# B&R Automation Studio project VInRoS_BaR_AS_Program
Automation Studio 4.12.5.95 SP; technology packages: mapp 5.24.2, mappCockpit 5.24.2, mappMotion 5.26.1, mappView 5.24.2

## Configuration Config_5APC2100

CPU 5APC2100.BY48-000, AutomationRuntime B4.83, Build 4.1.2, Safety 1.10, Vc V4.72.6

### Task classes (Cpu.sw)
```
Cyclic#1 (cycle 2000 us, tolerance 0 us):
  T_MECH_1 <- T_MECH_1.prg
  T_MECH_2 <- T_MECH_2.prg
  T_MECH_3 <- T_MECH_3.prg
Cyclic#2 (cycle 4000 us, tolerance 0 us):
  T_ROB_1 <- T_ROB_1.prg
  T_ROB_2_L <- T_ROB_2_L.prg
  T_ROB_2_R <- T_ROB_2_R.prg
Cyclic#3 (cycle 10000 us, tolerance 0 us):
  T_EX600 <- T_EX600.prg
DataObjects: assl1, McAcpSys
NcDataObjects: McDriveLog
Binaries: arsvcreg, FWRules, McAcpSim, mvLoader, mCoWebSc, McAcpDrv, TCData, udbdef, arflatprv, arcoal, iomap, asfw, Settings, Role, Cfg_mMot, sysconf, asnxdb1, arconfig, ashwac, ashwd, User, asnxdb2
Libraries: McBase, CoTrace, AsZip, FileIO, runtime, AsSafety, standard, DataObj, AsXml, astime, McAxis, McAcpAx, McAcpPar, McAxGroup, MpAxis, MpBase, arssl, powerlnk, asepl
```

### Hardware
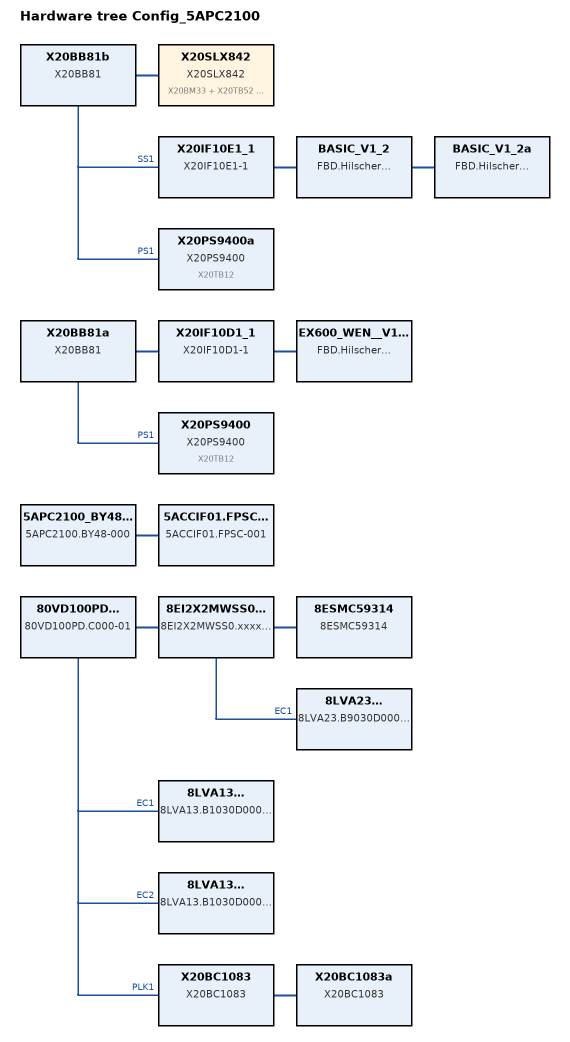
```
5ACCIF01.FPSC-001 : 5ACCIF01.FPSC-001 v1.9.1.0  [SL -> 5APC2100_BY48_000.SL1]
  Connector IF1:
    DNAConfiguration = manual
    Channel1
    ChannelID1 = McAcpBroadcast
    ChannelType1 = OCTET[128]
5APC2100_BY48_000 : 5APC2100.BY48-000 v2.1.1.0
  Connector IF3:
    AssignedOperatingSystem = ARemb
    ActivateDevice = 1
  Connector IF4:
    AssignedOperatingSystem = GPOS
  Connector IF7:
    OperatingSystem = ARemb
    ActivateDevice = 1
  Connector IF5:
    AssignedOperatingSystem = ARemb
  Connector IF6:
    AssignedOperatingSystem = GPOS
  ConfigurationID = BR_AS_I4C_Program_Config_5APC2100
  TimerDeviceType = EPLX2X
  TimerDevice = 5ACCIF01.FPSC-001.IF1
  TaskClassIdleTime = 2000
  Cyclic1Duration = 2000
  Cyclic1Tolerance = 0
  Cyclic2Duration = 4000
  Cyclic2Tolerance = 0
  Cyclic3Duration = 10000
  Cyclic3Tolerance = 0
  ActivateOpcUa = 1
  OpcUaInformationModels_PV_Version = 1
  ActivateHypervisor = 1
  ARembDramSizeInMb = 2000
80VD100PD.C000-01 : 80VD100PD.C000-01 v2.5.0.0  [PLK1 -> X20BC1083.PLK1 (NodeNumber=3) [Cable Type=PowerlinkCable, Length=10, Version=1.0.0.3]; PLK2 -> 8EI2X2MWSS0.xxxx-1.PLK1 (NodeNumber=3) [Cable Type=PowerlinkCable, Length=10, Version=1.0.0.3]; EC1 -> 8LVA13.B1030D000-0.EC; EC2 -> 8LVA13.B1030D000-0a.EC; MT2 -> 8LVA13.B1030D000-0a.MT]
  EnableDNA = on
  EPL_DNA_HubPort = 1
  DriveConfiguration/Module:
    McAcoposTypeID = AcoposMicroDConfig
    ActivateACOPOSSimulationOnPLC = 0
  DriveConfiguration/Channel[1]/RealAxis:
    AxisReference = gAxis_Mech_01
    MechanicalElementsIsInvisible = 0
  DriveConfiguration/Channel[1]/RealAxis/MechanicalElements/Gearbox:
    InputIsReadOnly = 0
    Input = 1
    OutputIsReadOnly = 0
    Output = 1
  DriveConfiguration/Channel[1]/RealAxis/MechanicalElements/RotaryToLinearTransformation:
    ReferenceDistanceIsReadOnly = 0
    ReferenceDistance = 54
  DriveConfiguration/Channel[1]/RealAxis/Controller:
    ModeIsReadOnly = 0
    Mode = PositionControllerWithTorqueFeedForward
  DriveConfiguration/Channel[1]/RealAxis/Controller/Mode/Position:
    ProportionalGainIsReadOnly = 0
    ProportionalGain = 279.0
    IntegrationTimeIsReadOnly = 0
    IntegrationTime = 0.000000
    TotalDelayTime = 0.0004
  DriveConfiguration/Channel[1]/RealAxis/Controller/Mode/Speed:
    ProportionalGainIsReadOnly = 0
    ProportionalGain = 0.25
    IntegrationTimeIsReadOnly = 0
    IntegrationTime = 0.000000
    FilterTimeIsReadOnly = 0
    FilterTime = 0.000000
  DriveConfiguration/Channel[1]/RealAxis/Controller/Mode:
    FeedForwardIsReadOnly = 0
    FeedForward = Standard
  DriveConfiguration/Channel[1]/RealAxis/Controller/Mode/FeedForward:
    TorqueLoad = 0.000000
    TorquePositive = 0.0326912
    TorqueNegative = 0.03062093
    SpeedTorqueFactor = 0.002517087
    Inertia = 0.00005712706
    AccelerationFilterTime = 0.000000
  DriveConfiguration/Channel[1]/RealAxis/Controller/Mode/LoopFilters:
    LoopFilterXIsReadOnly = 0
    LoopFilter1 = Notch
  DriveConfiguration/Channel[1]/RealAxis/Controller/Mode/LoopFilters/LoopFilter1:
    CenterFrequency = 166.3405
    Bandwidth = 400.000000
  DriveConfiguration/Channel[1]/RealAxis/Controller/Mode/LoopFilters:
    LoopFilter2 = NotUsed
    LoopFilter3 = NotUsed
  DriveConfiguration/Channel[1]/RealAxis/Homing:
    ModeIsReadOnly = 0
    Mode = Absolute
  DriveConfiguration/Channel[1]/RealAxis/Homing/Mode:
    Position = 1770365
  DriveConfiguration/Channel[1]/RealAxis/Homing:
    RestorePositionVariable = 
  DriveConfiguration/Channel[1]/RealAxis/StopReaction:
    QuickstopIsReadOnly = 0
    Quickstop = DecelerationLimit
    DriveErrorIsReadOnly = 0
    DriveError = DecelerationLimit
  DriveConfiguration/Channel[1]/RealAxis/MovementErrorLimits:
    PositionError = 1.0
    VelocityErrorMonitoring = Automatic1
  DriveConfiguration/Channel[1]/RealAxis:
    JerkFilterIsReadOnly = 0
    JerkFilter = Used
  DriveConfiguration/Channel[1]/RealAxis/JerkFilter:
    JerkTimeMin = 0
    JerkTime = 0.002
  DriveConfiguration/Channel[1]/RealAxis:
    ZeroVibrationFilter = NotUsed
  DriveConfiguration/Channel[1]/RealAxis/DigitalInputs/HomingSwitch:
    SourceIsReadOnly = 0
    Source = NotUsed
    Level = High
  DriveConfiguration/Channel[1]/RealAxis/DigitalInputs/PositiveLimitSwitch:
    SourceIsReadOnly = 0
    Source = NotUsed
    Level = High
  DriveConfiguration/Channel[1]/RealAxis/DigitalInputs/NegativeLimitSwitch:
    SourceIsReadOnly = 0
    Source = NotUsed
    Level = High
  DriveConfiguration/Channel[1]/RealAxis/DigitalInputs/Trigger1:
    Source = X2Trigger1
    Level = High
  DriveConfiguration/Channel[1]/RealAxis/DigitalInputs/Trigger2:
    Source = X2Trigger2
    Level = High
  DriveConfiguration/Channel[1]/RealAxis/DigitalInputs/Quickstop:
    Input = Trigger2
  DriveConfiguration/Channel[1]/RealAxis/Simulation:
    SimulationModeOnPLC = SetValueGeneration
    SimulationModeOnACOPOS = NotUsed
  DriveConfiguration/Channel[2]/RealAxis:
    AxisReference = gAxis_Mech_02
    MechanicalElementsIsInvisible = 0
  DriveConfiguration/Channel[2]/RealAxis/MechanicalElements/Gearbox:
    InputIsReadOnly = 0
    Input = 1
    OutputIsReadOnly = 0
    Output = 1
  DriveConfiguration/Channel[2]/RealAxis/MechanicalElements/RotaryToLinearTransformation:
    ReferenceDistanceIsReadOnly = 0
    ReferenceDistance = 54
  DriveConfiguration/Channel[2]/RealAxis/Controller:
    ModeIsReadOnly = 0
    Mode = PositionControllerWithTorqueFeedForward
  DriveConfiguration/Channel[2]/RealAxis/Controller/Mode/Position:
    ProportionalGainIsReadOnly = 0
    ProportionalGain = 282.0
    IntegrationTimeIsReadOnly = 0
    IntegrationTime = 0.000000
    TotalDelayTime = 0.000400
  DriveConfiguration/Channel[2]/RealAxis/Controller/Mode/Speed:
    ProportionalGainIsReadOnly = 0
    ProportionalGain = 0.25
    IntegrationTimeIsReadOnly = 0
    IntegrationTime = 0.000000
    FilterTimeIsReadOnly = 0
    FilterTime = 0.000000
  DriveConfiguration/Channel[2]/RealAxis/Controller/Mode:
    FeedForwardIsReadOnly = 0
    FeedForward = Standard
  DriveConfiguration/Channel[2]/RealAxis/Controller/Mode/FeedForward:
    TorqueLoad = 0.000000
    TorquePositive = 0.03686025
    TorqueNegative = 0.03496668
    SpeedTorqueFactor = 0.002854001
    Inertia = 0.00005443416
    AccelerationFilterTime = 0.000000
  DriveConfiguration/Channel[2]/RealAxis/Controller/Mode/LoopFilters:
    LoopFilterXIsReadOnly = 0
    LoopFilter1 = Notch
  DriveConfiguration/Channel[2]/RealAxis/Controller/Mode/LoopFilters/LoopFilter1:
    CenterFrequency = 176.1253
    Bandwidth = 400.000000
  DriveConfiguration/Channel[2]/RealAxis/Controller/Mode/LoopFilters:
    LoopFilter2 = NotUsed
    LoopFilter3 = NotUsed
  DriveConfiguration/Channel[2]/RealAxis/Homing:
    ModeIsReadOnly = 0
    Mode = Absolute
  DriveConfiguration/Channel[2]/RealAxis/Homing/Mode:
    Position = 2219977
  DriveConfiguration/Channel[2]/RealAxis/Homing:
    RestorePositionVariable = 
  DriveConfiguration/Channel[2]/RealAxis/StopReaction:
    QuickstopIsReadOnly = 0
    Quickstop = DecelerationLimit
    DriveErrorIsReadOnly = 0
    DriveError = DecelerationLimit
  DriveConfiguration/Channel[2]/RealAxis/MovementErrorLimits:
    PositionError = 1.0
    VelocityErrorMonitoring = Automatic1
  DriveConfiguration/Channel[2]/RealAxis:
    JerkFilterIsReadOnly = 0
    JerkFilter = Used
  DriveConfiguration/Channel[2]/RealAxis/JerkFilter:
    JerkTimeMin = 0
    JerkTime = 0.002
  DriveConfiguration/Channel[2]/RealAxis:
    ZeroVibrationFilter = NotUsed
  DriveConfiguration/Channel[2]/RealAxis/DigitalInputs/HomingSwitch:
    SourceIsReadOnly = 0
    Source = NotUsed
    Level = High
  DriveConfiguration/Channel[2]/RealAxis/DigitalInputs/PositiveLimitSwitch:
    SourceIsReadOnly = 0
    Source = NotUsed
    Level = High
  DriveConfiguration/Channel[2]/RealAxis/DigitalInputs/NegativeLimitSwitch:
    SourceIsReadOnly = 0
    Source = NotUsed
    Level = High
  DriveConfiguration/Channel[2]/RealAxis/DigitalInputs/Trigger1:
    Source = X2Trigger1
    Level = High
  DriveConfiguration/Channel[2]/RealAxis/DigitalInputs/Trigger2:
    Source = X2Trigger2
    Level = High
  DriveConfiguration/Channel[2]/RealAxis/DigitalInputs/Quickstop:
    Input = Trigger2
  DriveConfiguration/Channel[2]/RealAxis/Simulation:
    SimulationModeOnPLC = SetValueGeneration
    SimulationModeOnACOPOS = NotUsed
8EI2X2MWSS0.xxxx-1 : 8EI2X2MWSS0.xxxx-1 v2.4.0.1  [PLK1 -> 80VD100PD.C000-01.PLK2 (NodeNumber=4) [Cable Type=PowerlinkCable, Length=10, Version=1.0.0.3]; EC1 -> 8LVA23.B9030D000-0.EC]
  EnableDNA = on
  EPL_DNA_Head = 0
  EPL_DNA_Predecessor = 3
  EPL_DNA_InPort = 2
  McAcpModuleTypeID = AcoposP3SafeMotion
  DriveConfiguration/Module:
    McAcoposTypeID = AcoposP3SConfig
    ActivateACOPOSSimulationOnPLC = 0
  DriveConfiguration/Channel[1]/RealAxis:
    AxisReference = gAxis_Mech_03
    MechanicalElementsIsInvisible = 0
  DriveConfiguration/Channel[1]/RealAxis/MechanicalElements/Gearbox:
    InputIsReadOnly = 0
    Input = 1
    OutputIsReadOnly = 0
    Output = 1
  DriveConfiguration/Channel[1]/RealAxis/MechanicalElements/RotaryToLinearTransformation:
    ReferenceDistanceIsReadOnly = 0
    ReferenceDistance = 20
  DriveConfiguration/Channel[1]/RealAxis/Controller:
    ModeIsReadOnly = 0
    Mode = PositionControllerWithTorqueFeedForward
  DriveConfiguration/Channel[1]/RealAxis/Controller/Mode/Position:
    ProportionalGainIsReadOnly = 0
    ProportionalGain = 340
    IntegrationTimeIsReadOnly = 0
    IntegrationTime = 0.0
    TotalDelayTime = 0.0004
  DriveConfiguration/Channel[1]/RealAxis/Controller/Mode/Speed:
    ProportionalGainIsReadOnly = 0
    ProportionalGain = 3.8
    IntegrationTimeIsReadOnly = 0
    IntegrationTime = 0.0
    FilterTimeIsReadOnly = 0
    FilterTime = 0.0
  DriveConfiguration/Channel[1]/RealAxis/Controller/Mode:
    FeedForwardIsReadOnly = 0
    FeedForward = Standard
  DriveConfiguration/Channel[1]/RealAxis/Controller/Mode/FeedForward:
    TorqueLoad = 0.0
    TorquePositive = 0.1956726
    TorqueNegative = 0.1982097
    SpeedTorqueFactor = 0.0
    Inertia = 0.0
    AccelerationFilterTime = 0.0
  DriveConfiguration/Channel[1]/RealAxis/Controller/Mode/LoopFilters:
    LoopFilterXIsReadOnly = 0
    LoopFilter1 = Notch
  DriveConfiguration/Channel[1]/RealAxis/Controller/Mode/LoopFilters/LoopFilter1:
    CenterFrequency = 2181.996
    Bandwidth = 400
  DriveConfiguration/Channel[1]/RealAxis/Controller/Mode/LoopFilters:
    LoopFilter2 = NotUsed
    LoopFilter3 = NotUsed
  DriveConfiguration/Channel[1]/RealAxis/Homing:
    ModeIsReadOnly = 0
    Mode = Absolute
  DriveConfiguration/Channel[1]/RealAxis/Homing/Mode:
    Position = -21168.21
  DriveConfiguration/Channel[1]/RealAxis/Homing:
    RestorePositionVariable = 
  DriveConfiguration/Channel[1]/RealAxis/StopReaction:
    QuickstopIsReadOnly = 0
    Quickstop = DecelerationLimit
    DriveErrorIsReadOnly = 0
    DriveError = DecelerationLimit
  DriveConfiguration/Channel[1]/RealAxis/MovementErrorLimits:
    PositionError = 1
    VelocityErrorMonitoring = Automatic1
  DriveConfiguration/Channel[1]/RealAxis:
    JerkFilterIsReadOnly = 0
    JerkFilter = Used
  DriveConfiguration/Channel[1]/RealAxis/JerkFilter:
    JerkTimeMin = 0
    JerkTime = 0.002
  DriveConfiguration/Channel[1]/RealAxis:
    ZeroVibrationFilter = NotUsed
  DriveConfiguration/Channel[1]/RealAxis/DigitalInputs/HomingSwitch:
    SourceIsReadOnly = 0
    Source = NotUsed
    Level = High
  DriveConfiguration/Channel[1]/RealAxis/DigitalInputs/PositiveLimitSwitch:
    SourceIsReadOnly = 0
    Source = NotUsed
    Level = High
  DriveConfiguration/Channel[1]/RealAxis/DigitalInputs/NegativeLimitSwitch:
    SourceIsReadOnly = 0
    Source = NotUsed
    Level = High
  DriveConfiguration/Channel[1]/RealAxis/DigitalInputs/Trigger1:
    Source = X8Trigger1
    Level = High
  DriveConfiguration/Channel[1]/RealAxis/DigitalInputs/Trigger2:
    Source = X8Trigger2
    Level = High
  DriveConfiguration/Channel[1]/RealAxis/DigitalInputs/Quickstop:
    Input = NotUsed
  DriveConfiguration/Channel[1]/RealAxis/Simulation:
    SimulationModeOnPLC = SetValueGeneration
    SimulationModeOnACOPOS = NotUsed
  DriveConfiguration/Channel[1]:
    ExternalEncoderAxis = NotUsed
8ESMC59314 : 8ESMC59314 v1.10.3.1  [SafeMOTION -> 8EI2X2MWSS0.xxxx-1.SafeMOTION1]
8LVA13.B1030D000-0 : 8LVA13.B1030D000-0 v2.2.0.3  [EC -> 80VD100PD.C000-01.EC1; MT -> 80VD100PD.C000-01.MT1]
  M1/MotorParameters:
    MOTOR_AMB_TEMP_RATED = 40
8LVA13.B1030D000-0a : 8LVA13.B1030D000-0 v2.2.0.3  [EC -> 80VD100PD.C000-01.EC2; MT -> 80VD100PD.C000-01.MT2]
  M1/MotorParameters:
    MOTOR_AMB_TEMP_RATED = 40
8LVA23.B9030D000-0 : 8LVA23.B9030D000-0 v2.2.0.3  [EC -> 8EI2X2MWSS0.xxxx-1.EC1; MT -> 8EI2X2MWSS0.xxxx-1.MT1]
  M1/MotorParameters:
    MOTOR_AMB_TEMP_RATED = 40
BASIC_V1_2 : FBD.Hilscher.PNIOGenDevDTM2.BASIC V1.2 v1.2 (OrderNumber=BASIC V1.2, VendorAddress=irb120)  [PN1 -> X20IF10E1_1.IF1]
  DtmId = f66cc699-ca5c-46ca-9c78-189869e182c2
BASIC_V1_2a : FBD.Hilscher.PNIOGenDevDTM2.BASIC V1.2 v1.2 (OrderNumber=BASIC V1.2, VendorAddress=irb14000)  [PN1 -> BASIC_V1_2.PN2]
  DtmId = 47b40347-aff1-415b-a34d-ab04019bc4a6
  ChannelBlocks_bb3f4ff7-7be2-449f-96d3-48042bfc087e  // DI 256 bytes <Slot 1>
  IO_InputImage_bb3f4ff7-7be2-449f-96d3-48042bfc087e  // 256 Byte(s)
  ChannelBlocks_57420719-53a5-465f-bb9f-9beb1182c40e  // DO 256 bytes <Slot 2>
  IO_OutputImage_57420719-53a5-465f-bb9f-9beb1182c40e  // 256 Byte(s)
EX600_WEN__V1_1 : FBD.Hilscher.EIGenEDSAdapterDTM.EX600-WEN$002A V1.1 v1.1 (OrderNumber=EX600-WEN* V1.1, VendorAddress=192.168.123.3)  [EIP1 -> X20IF10D1_1.IF1]
  DtmId = fe5fa07e-a34a-4bd5-a4b6-be2963ba3a9e
  ChannelBlocks_b68dcd95-6382-41a2-8458-d2ed95ac6e1a  // Module 0
  IO_InputImage_b68dcd95-6382-41a2-8458-d2ed95ac6e1a  // 12 Byte(s)
  IO_OutputImage_b68dcd95-6382-41a2-8458-d2ed95ac6e1a  // 4 Byte(s)
X20BB81a : X20BB81 v1.2.0.0
X20BB81b : X20BB81 v1.2.0.0
X20BC1083 : X20BC1083 v2.14.0.0  [PLK1 -> 80VD100PD.C000-01.PLK1 (NodeNumber=2) [Cable Type=PowerlinkCable, Length=10, Version=1.0.0.3]; PLK2 -> X20BC1083a.PLK1 (NodeNumber=2) [Cable Type=PowerlinkCable, Length=10, Version=1.0.0.3]; SL -> X20BB81b.SL1]
X20BC1083a : X20BC1083 v2.14.0.0  [PLK1 -> X20BC1083.PLK2 (NodeNumber=1) [Cable Type=PowerlinkCable, Length=10, Version=1.0.0.3]; PLK2 -> 5ACCIF01.FPSC-001.IF1 (NodeNumber=1) [Cable Type=PowerlinkCable, Length=10, Version=1.0.0.3]; SL -> X20BB81a.SL1]
  Supervision = off
X20BM33a : X20BM33 v1.1.0.0  [X2X1 -> X20BB81b.IF1]
X20IF10D1_1 : X20IF10D1-1 v1.7.0.0  [SS -> X20BB81a.SS1]
  Connector IF1:
    DtmId = 7208ef1e-b1a4-4925-887c-724f10ed4697
  ConfigFile = X20IF10D1_1.dtm
  ConfigModule = asnxdb1
X20IF10E1_1 : X20IF10E1-1 v1.4.0.0  [SS -> X20BB81b.SS1]
  Connector IF1:
    DtmId = d38f4261-e439-4a9b-81eb-d6637cfccb7f
  ConfigFile = X20IF10E1_1.dtm
  ConfigModule = asnxdb2
  CycleTime = 4000
X20PS9400 : X20PS9400 v1.8.0.0  [SS1 -> X20TB12.SS; PS -> X20BB81a.PS1]
X20PS9400a : X20PS9400 v1.8.0.0  [SS1 -> X20TB12a.SS; PS -> X20BB81b.PS1]
X20SLX842 : X20SLX842 v1.10.12.1  [SS1 -> X20TB52.SS; SS2 -> X20TB52a.SS; SL -> X20BM33a.SL1]
  SafeProject = SafeLOGIC-1
  SafeDesigner = 4.4.1.0
X20TB12 : X20TB12 v1.0.0.0
X20TB12a : X20TB12 v1.0.0.0
X20TB52 : X20TB52 v1.0.0.2
X20TB52a : X20TB52 v1.0.0.2
```

### IoMap.iom - 5APC2100_BY48_000/IoMap.iom
```iecst
VAR_CONFIG
	::RESET_SAFETY AT %QX."X20SLX842".BOOL101;
	::Global_VInRoS_Str.EX_600.Slave.Info.Active AT %IX."EX600_WEN__V1_1".ModuleOk;
	::T_EX600:C_USINT_To_BOOL_Arr_1.INPUT AT %IB."EX600_WEN__V1_1".Module_0_Input011;
	::T_EX600:C_USINT_To_BOOL_Arr_2.INPUT AT %IB."EX600_WEN__V1_1".Module_0_Input012;
	::T_EX600:C_BOOL_Arr_To_USINT_1.OUTPUT AT %QB."EX600_WEN__V1_1".Module_0_Output003;
	::SAFETY_ACTIVE AT %IX."X20SLX842".SafeDigitalInput03;
	::SAFETY_STATUS AT %IX."X20SLX842".BOOL001;
	::T_ROB_1:ABB_Library_Rob_1.Status.PLC.Module_OK AT %IX."BASIC_V1_2".ModuleOk;
	::T_ROB_1:ABB_Library_Rob_1.PROFINET_Mapping_IN.STATUS.INPUT AT %IB."BASIC_V1_2".Module001_Input_0;
	::T_ROB_1:ABB_Library_Rob_1.PROFINET_Mapping_IN.SYSTEM.INPUT AT %IB."BASIC_V1_2".Module001_Input_1;
	::T_ROB_1:ABB_Library_Rob_1.PROFINET_Mapping_IN.STATE_uID AT %IB."BASIC_V1_2".Module001_Input_2;
	::T_ROB_1:ABB_Library_Rob_1.PROFINET_Mapping_IN.STATE_mID AT %IB."BASIC_V1_2".Module001_Input_3;
	::T_ROB_1:ABB_Library_Rob_1.PROFINET_Mapping_IN.MOTION_TRAJECTORY_ID.INPUT[0] AT %IB."BASIC_V1_2".Module001_Input_4;
	::T_ROB_1:ABB_Library_Rob_1.PROFINET_Mapping_IN.MOTION_TRAJECTORY_ID.INPUT[1] AT %IB."BASIC_V1_2".Module001_Input_5;
	::T_ROB_1:ABB_Library_Rob_1.PROFINET_Mapping_IN.JOINT_POS[0].INPUT[0] AT %IB."BASIC_V1_2".Module001_Input_6;
	::T_ROB_1:ABB_Library_Rob_1.PROFINET_Mapping_IN.JOINT_POS[0].INPUT[1] AT %IB."BASIC_V1_2".Module001_Input_7;
	::T_ROB_1:ABB_Library_Rob_1.PROFINET_Mapping_IN.JOINT_POS[1].INPUT[0] AT %IB."BASIC_V1_2".Module001_Input_8;
	::T_ROB_1:ABB_Library_Rob_1.PROFINET_Mapping_IN.JOINT_POS[1].INPUT[1] AT %IB."BASIC_V1_2".Module001_Input_9;
	::T_ROB_1:ABB_Library_Rob_1.PROFINET_Mapping_IN.JOINT_POS[2].INPUT[0] AT %IB."BASIC_V1_2".Module001_Input_10;
	::T_ROB_1:ABB_Library_Rob_1.PROFINET_Mapping_IN.JOINT_POS[2].INPUT[1] AT %IB."BASIC_V1_2".Module001_Input_11;
	::T_ROB_1:ABB_Library_Rob_1.PROFINET_Mapping_IN.JOINT_POS[3].INPUT[0] AT %IB."BASIC_V1_2".Module001_Input_12;
	::T_ROB_1:ABB_Library_Rob_1.PROFINET_Mapping_IN.JOINT_POS[3].INPUT[1] AT %IB."BASIC_V1_2".Module001_Input_13;
	::T_ROB_1:ABB_Library_Rob_1.PROFINET_Mapping_IN.JOINT_POS[4].INPUT[0] AT %IB."BASIC_V1_2".Module001_Input_14;
	::T_ROB_1:ABB_Library_Rob_1.PROFINET_Mapping_IN.JOINT_POS[4].INPUT[1] AT %IB."BASIC_V1_2".Module001_Input_15;
	::T_ROB_1:ABB_Library_Rob_1.PROFINET_Mapping_IN.JOINT_POS[5].INPUT[0] AT %IB."BASIC_V1_2".Module001_Input_16;
	::T_ROB_1:ABB_Library_Rob_1.PROFINET_Mapping_IN.JOINT_POS[5].INPUT[1] AT %IB."BASIC_V1_2".Module001_Input_17;
	::T_ROB_1:ABB_Library_Rob_1.PROFINET_Mapping_IN.JOINT_POS[6].INPUT[0] AT %IB."BASIC_V1_2".Module001_Input_18;
	::T_ROB_1:ABB_Library_Rob_1.PROFINET_Mapping_IN.JOINT_POS[6].INPUT[1] AT %IB."BASIC_V1_2".Module001_Input_19;
	::T_ROB_1:ABB_Library_Rob_1.PROFINET_Mapping_IN.JOINT_POS_SIGN.INPUT AT %IB."BASIC_V1_2".Module001_Input_20;
	::T_ROB_1:ABB_Library_Rob_1.PROFINET_Mapping_IN.TCP_POS[0].INPUT[0] AT %IB."BASIC_V1_2".Module001_Input_21;
	::T_ROB_1:ABB_Library_Rob_1.PROFINET_Mapping_IN.TCP_POS[0].INPUT[1] AT %IB."BASIC_V1_2".Module001_Input_22;
	::T_ROB_1:ABB_Library_Rob_1.PROFINET_Mapping_IN.TCP_POS[0].INPUT[2] AT %IB."BASIC_V1_2".Module001_Input_23;
	::T_ROB_1:ABB_Library_Rob_1.PROFINET_Mapping_IN.TCP_POS[0].INPUT[3] AT %IB."BASIC_V1_2".Module001_Input_24;
	::T_ROB_1:ABB_Library_Rob_1.PROFINET_Mapping_IN.TCP_POS[1].INPUT[0] AT %IB."BASIC_V1_2".Module001_Input_25;
	::T_ROB_1:ABB_Library_Rob_1.PROFINET_Mapping_IN.TCP_POS[1].INPUT[1] AT %IB."BASIC_V1_2".Module001_Input_26;
	::T_ROB_1:ABB_Library_Rob_1.PROFINET_Mapping_IN.TCP_POS[1].INPUT[2] AT %IB."BASIC_V1_2".Module001_Input_27;
	::T_ROB_1:ABB_Library_Rob_1.PROFINET_Mapping_IN.TCP_POS[1].INPUT[3] AT %IB."BASIC_V1_2".Module001_Input_28;
	::T_ROB_1:ABB_Library_Rob_1.PROFINET_Mapping_IN.TCP_POS[2].INPUT[0] AT %IB."BASIC_V1_2".Module001_Input_29;
	::T_ROB_1:ABB_Library_Rob_1.PROFINET_Mapping_IN.TCP_POS[2].INPUT[1] AT %IB."BASIC_V1_2".Module001_Input_30;
	::T_ROB_1:ABB_Library_Rob_1.PROFINET_Mapping_IN.TCP_POS[2].INPUT[2] AT %IB."BASIC_V1_2".Module001_Input_31;
	::T_ROB_1:ABB_Library_Rob_1.PROFINET_Mapping_IN.TCP_POS[2].INPUT[3] AT %IB."BASIC_V1_2".Module001_Input_32;
	::T_ROB_1:ABB_Library_Rob_1.PROFINET_Mapping_IN.TCP_ROT[0].INPUT[0] AT %IB."BASIC_V1_2".Module001_Input_33;
	::T_ROB_1:ABB_Library_Rob_1.PROFINET_Mapping_IN.TCP_ROT[0].INPUT[1] AT %IB."BASIC_V1_2".Module001_Input_34;
	::T_ROB_1:ABB_Library_Rob_1.PROFINET_Mapping_IN.TCP_ROT[1].INPUT[0] AT %IB."BASIC_V1_2".Module001_Input_35;
	::T_ROB_1:ABB_Library_Rob_1.PROFINET_Mapping_IN.TCP_ROT[1].INPUT[1] AT %IB."BASIC_V1_2".Module001_Input_36;
	::T_ROB_1:ABB_Library_Rob_1.PROFINET_Mapping_IN.TCP_ROT[2].INPUT[0] AT %IB."BASIC_V1_2".Module001_Input_37;
	::T_ROB_1:ABB_Library_Rob_1.PROFINET_Mapping_IN.TCP_ROT[2].INPUT[1] AT %IB."BASIC_V1_2".Module001_Input_38;
	::T_ROB_1:ABB_Library_Rob_1.PROFINET_Mapping_IN.TCP_EX_POS.INPUT[0] AT %IB."BASIC_V1_2".Module001_Input_39;
	::T_ROB_1:ABB_Library_Rob_1.PROFINET_Mapping_IN.TCP_EX_POS.INPUT[1] AT %IB."BASIC_V1_2".Module001_Input_40;
	::T_ROB_1:ABB_Library_Rob_1.PROFINET_Mapping_IN.TCP_SIGN.INPUT AT %IB."BASIC_V1_2".Module001_Input_41;
	::T_ROB_1:ABB_Library_Rob_1.PROFINET_Mapping_IN.TCP_CFG[0] AT %IB."BASIC_V1_2".Module001_Input_42;
	::T_ROB_1:ABB_Library_Rob_1.PROFINET_Mapping_IN.TCP_CFG[1] AT %IB."BASIC_V1_2".Module001_Input_43;
	::T_ROB_1:ABB_Library_Rob_1.PROFINET_Mapping_IN.TCP_CFG[2] AT %IB."BASIC_V1_2".Module001_Input_44;
	::T_ROB_1:ABB_Library_Rob_1.PROFINET_Mapping_IN.TCP_CFG[3] AT %IB."BASIC_V1_2".Module001_Input_45;
	::T_ROB_1:ABB_Library_Rob_1.PROFINET_Mapping_IN.TCP_CFG_SIGN.INPUT AT %IB."BASIC_V1_2".Module001_Input_46;
	::T_ROB_1:ABB_Library_Rob_1.PROFINET_Mapping_OUT.STATUS.OUTPUT AT %QB."BASIC_V1_2".Module002_Output_0;
	::T_ROB_1:ABB_Library_Rob_1.PROFINET_Mapping_OUT.SYSTEM.OUTPUT AT %QB."BASIC_V1_2".Module002_Output_1;
	::T_ROB_1:ABB_Library_Rob_1.PROFINET_Mapping_OUT.COMMAND.OUTPUT AT %QB."BASIC_V1_2".Module002_Output_2;
	::T_ROB_1:ABB_Library_Rob_1.PROFINET_Mapping_OUT.COMMAND_mID AT %QB."BASIC_V1_2".Module002_Output_3;
	::T_ROB_1:ABB_Library_Rob_1.PROFINET_Mapping_OUT.COMMAND_uID AT %QB."BASIC_V1_2".Module002_Output_4;
	::T_ROB_1:ABB_Library_Rob_1.PROFINET_Mapping_OUT.TRAJECTORY_SIZE.OUTPUT[0] AT %QB."BASIC_V1_2".Module002_Output_5;
	::T_ROB_1:ABB_Library_Rob_1.PROFINET_Mapping_OUT.TRAJECTORY_SIZE.OUTPUT[1] AT %QB."BASIC_V1_2".Module002_Output_6;
	::T_ROB_1:ABB_Library_Rob_1.PROFINET_Mapping_OUT.SPEED AT %QB."BASIC_V1_2".Module002_Output_7;
	::T_ROB_1:ABB_Library_Rob_1.PROFINET_Mapping_OUT.ZONE AT %QB."BASIC_V1_2".Module002_Output_8;
	::T_ROB_1:ABB_Library_Rob_1.PROFINET_Mapping_OUT.JOINT_POS[0].OUTPUT[0] AT %QB."BASIC_V1_2".Module002_Output_9;
	::T_ROB_1:ABB_Library_Rob_1.PROFINET_Mapping_OUT.JOINT_POS[0].OUTPUT[1] AT %QB."BASIC_V1_2".Module002_Output_10;
	::T_ROB_1:ABB_Library_Rob_1.PROFINET_Mapping_OUT.JOINT_POS[1].OUTPUT[0] AT %QB."BASIC_V1_2".Module002_Output_11;
	::T_ROB_1:ABB_Library_Rob_1.PROFINET_Mapping_OUT.JOINT_POS[1].OUTPUT[1] AT %QB."BASIC_V1_2".Module002_Output_12;
	::T_ROB_1:ABB_Library_Rob_1.PROFINET_Mapping_OUT.JOINT_POS[2].OUTPUT[0] AT %QB."BASIC_V1_2".Module002_Output_13;
	::T_ROB_1:ABB_Library_Rob_1.PROFINET_Mapping_OUT.JOINT_POS[2].OUTPUT[1] AT %QB."BASIC_V1_2".Module002_Output_14;
	::T_ROB_1:ABB_Library_Rob_1.PROFINET_Mapping_OUT.JOINT_POS[3].OUTPUT[0] AT %QB."BASIC_V1_2".Module002_Output_15;
	::T_ROB_1:ABB_Library_Rob_1.PROFINET_Mapping_OUT.JOINT_POS[3].OUTPUT[1] AT %QB."BASIC_V1_2".Module002_Output_16;
	::T_ROB_1:ABB_Library_Rob_1.PROFINET_Mapping_OUT.JOINT_POS[4].OUTPUT[0] AT %QB."BASIC_V1_2".Module002_Output_17;
	::T_ROB_1:ABB_Library_Rob_1.PROFINET_Mapping_OUT.JOINT_POS[4].OUTPUT[1] AT %QB."BASIC_V1_2".Module002_Output_18;
	::T_ROB_1:ABB_Library_Rob_1.PROFINET_Mapping_OUT.JOINT_POS[5].OUTPUT[0] AT %QB."BASIC_V1_2".Module002_Output_19;
	::T_ROB_1:ABB_Library_Rob_1.PROFINET_Mapping_OUT.JOINT_POS[5].OUTPUT[1] AT %QB."BASIC_V1_2".Module002_Output_20;
	::T_ROB_1:ABB_Library_Rob_1.PROFINET_Mapping_OUT.JOINT_POS[6].OUTPUT[0] AT %QB."BASIC_V1_2".Module002_Output_21;
	::T_ROB_1:ABB_Library_Rob_1.PROFINET_Mapping_OUT.JOINT_POS[6].OUTPUT[1] AT %QB."BASIC_V1_2".Module002_Output_22;
	::T_ROB_1:ABB_Library_Rob_1.PROFINET_Mapping_OUT.JOINT_POS_SIGN.OUTPUT AT %QB."BASIC_V1_2".Module002_Output_23;
	::T_ROB_1:ABB_Library_Rob_1.PROFINET_Mapping_OUT.TCP_POS[0].OUTPUT[0] AT %QB."BASIC_V1_2".Module002_Output_24;
	::T_ROB_1:ABB_Library_Rob_1.PROFINET_Mapping_OUT.TCP_POS[0].OUTPUT[1] AT %QB."BASIC_V1_2".Module002_Output_25;
	::T_ROB_1:ABB_Library_Rob_1.PROFINET_Mapping_OUT.TCP_POS[0].OUTPUT[2] AT %QB."BASIC_V1_2".Module002_Output_26;
	::T_ROB_1:ABB_Library_Rob_1.PROFINET_Mapping_OUT.TCP_POS[0].OUTPUT[3] AT %QB."BASIC_V1_2".Module002_Output_27;
	::T_ROB_1:ABB_Library_Rob_1.PROFINET_Mapping_OUT.TCP_POS[1].OUTPUT[0] AT %QB."BASIC_V1_2".Module002_Output_28;
	::T_ROB_1:ABB_Library_Rob_1.PROFINET_Mapping_OUT.TCP_POS[1].OUTPUT[1] AT %QB."BASIC_V1_2".Module002_Output_29;
	::T_ROB_1:ABB_Library_Rob_1.PROFINET_Mapping_OUT.TCP_POS[1].OUTPUT[2] AT %QB."BASIC_V1_2".Module002_Output_30;
	::T_ROB_1:ABB_Library_Rob_1.PROFINET_Mapping_OUT.TCP_POS[1].OUTPUT[3] AT %QB."BASIC_V1_2".Module002_Output_31;
	::T_ROB_1:ABB_Library_Rob_1.PROFINET_Mapping_OUT.TCP_POS[2].OUTPUT[0] AT %QB."BASIC_V1_2".Module002_Output_32;
	::T_ROB_1:ABB_Library_Rob_1.PROFINET_Mapping_OUT.TCP_POS[2].OUTPUT[1] AT %QB."BASIC_V1_2".Module002_Output_33;
	::T_ROB_1:ABB_Library_Rob_1.PROFINET_Mapping_OUT.TCP_POS[2].OUTPUT[2] AT %QB."BASIC_V1_2".Module002_Output_34;
	::T_ROB_1:ABB_Library_Rob_1.PROFINET_Mapping_OUT.TCP_POS[2].OUTPUT[3] AT %QB."BASIC_V1_2".Module002_Output_35;
	::T_ROB_1:ABB_Library_Rob_1.PROFINET_Mapping_OUT.TCP_ROT[0].OUTPUT[0] AT %QB."BASIC_V1_2".Module002_Output_36;
	::T_ROB_1:ABB_Library_Rob_1.PROFINET_Mapping_OUT.TCP_ROT[0].OUTPUT[1] AT %QB."BASIC_V1_2".Module002_Output_37;
	::T_ROB_1:ABB_Library_Rob_1.PROFINET_Mapping_OUT.TCP_ROT[1].OUTPUT[0] AT %QB."BASIC_V1_2".Module002_Output_38;
	::T_ROB_1:ABB_Library_Rob_1.PROFINET_Mapping_OUT.TCP_ROT[1].OUTPUT[1] AT %QB."BASIC_V1_2".Module002_Output_39;
	::T_ROB_1:ABB_Library_Rob_1.PROFINET_Mapping_OUT.TCP_ROT[2].OUTPUT[0] AT %QB."BASIC_V1_2".Module002_Output_40;
	::T_ROB_1:ABB_Library_Rob_1.PROFINET_Mapping_OUT.TCP_ROT[2].OUTPUT[1] AT %QB."BASIC_V1_2".Module002_Output_41;
	::T_ROB_1:ABB_Library_Rob_1.PROFINET_Mapping_OUT.TCP_EX_POS.OUTPUT[0] AT %QB."BASIC_V1_2".Module002_Output_42;
	::T_ROB_1:ABB_Library_Rob_1.PROFINET_Mapping_OUT.TCP_EX_POS.OUTPUT[1] AT %QB."BASIC_V1_2".Module002_Output_43;
	::T_ROB_1:ABB_Library_Rob_1.PROFINET_Mapping_OUT.TCP_SIGN.OUTPUT AT %QB."BASIC_V1_2".Module002_Output_44;
	::T_ROB_1:ABB_Library_Rob_1.PROFINET_Mapping_OUT.TCP_CFG[0] AT %QB."BASIC_V1_2".Module002_Output_45;
	::T_ROB_1:ABB_Library_Rob_1.PROFINET_Mapping_OUT.TCP_CFG[1] AT %QB."BASIC_V1_2".Module002_Output_46;
	::T_ROB_1:ABB_Library_Rob_1.PROFINET_Mapping_OUT.TCP_CFG[2] AT %QB."BASIC_V1_2".Module002_Output_47;
	::T_ROB_1:ABB_Library_Rob_1.PROFINET_Mapping_OUT.TCP_CFG[3] AT %QB."BASIC_V1_2".Module002_Output_48;
	::T_ROB_1:ABB_Library_Rob_1.PROFINET_Mapping_OUT.TCP_CFG_SIGN.OUTPUT AT %QB."BASIC_V1_2".Module002_Output_49;
	::T_ROB_1:ABB_Library_Rob_1.PROFINET_Mapping_OUT.RTOOL_RH.OUTPUT AT %QB."BASIC_V1_2".Module002_Output_50;
	::T_ROB_1:ABB_Library_Rob_1.PROFINET_Mapping_OUT.RTOOL_POS[0].OUTPUT[0] AT %QB."BASIC_V1_2".Module002_Output_51;
	::T_ROB_1:ABB_Library_Rob_1.PROFINET_Mapping_OUT.RTOOL_POS[0].OUTPUT[1] AT %QB."BASIC_V1_2".Module002_Output_52;
	::T_ROB_1:ABB_Library_Rob_1.PROFINET_Mapping_OUT.RTOOL_POS[1].OUTPUT[0] AT %QB."BASIC_V1_2".Module002_Output_53;
	::T_ROB_1:ABB_Library_Rob_1.PROFINET_Mapping_OUT.RTOOL_POS[1].OUTPUT[1] AT %QB."BASIC_V1_2".Module002_Output_54;
	::T_ROB_1:ABB_Library_Rob_1.PROFINET_Mapping_OUT.RTOOL_POS[2].OUTPUT[0] AT %QB."BASIC_V1_2".Module002_Output_55;
	::T_ROB_1:ABB_Library_Rob_1.PROFINET_Mapping_OUT.RTOOL_POS[2].OUTPUT[1] AT %QB."BASIC_V1_2".Module002_Output_56;
	::T_ROB_1:ABB_Library_Rob_1.PROFINET_Mapping_OUT.RTOOL_POS_SIGN.OUTPUT AT %QB."BASIC_V1_2".Module002_Output_57;
	::T_ROB_1:ABB_Library_Rob_1.PROFINET_Mapping_OUT.RTOOL_ROT_QUAT[0].OUTPUT[0] AT %QB."BASIC_V1_2".Module002_Output_58;
	::T_ROB_1:ABB_Library_Rob_1.PROFINET_Mapping_OUT.RTOOL_ROT_QUAT[0].OUTPUT[1] AT %QB."BASIC_V1_2".Module002_Output_59;
	::T_ROB_1:ABB_Library_Rob_1.PROFINET_Mapping_OUT.RTOOL_ROT_QUAT[0].OUTPUT[2] AT %QB."BASIC_V1_2".Module002_Output_60;
	::T_ROB_1:ABB_Library_Rob_1.PROFINET_Mapping_OUT.RTOOL_ROT_QUAT[0].OUTPUT[3] AT %QB."BASIC_V1_2".Module002_Output_61;
	::T_ROB_1:ABB_Library_Rob_1.PROFINET_Mapping_OUT.RTOOL_ROT_QUAT[1].OUTPUT[0] AT %QB."BASIC_V1_2".Module002_Output_62;
	::T_ROB_1:ABB_Library_Rob_1.PROFINET_Mapping_OUT.RTOOL_ROT_QUAT[1].OUTPUT[1] AT %QB."BASIC_V1_2".Module002_Output_63;
	::T_ROB_1:ABB_Library_Rob_1.PROFINET_Mapping_OUT.RTOOL_ROT_QUAT[1].OUTPUT[2] AT %QB."BASIC_V1_2".Module002_Output_64;
	::T_ROB_1:ABB_Library_Rob_1.PROFINET_Mapping_OUT.RTOOL_ROT_QUAT[1].OUTPUT[3] AT %QB."BASIC_V1_2".Module002_Output_65;
	::T_ROB_1:ABB_Library_Rob_1.PROFINET_Mapping_OUT.RTOOL_ROT_QUAT[2].OUTPUT[0] AT %QB."BASIC_V1_2".Module002_Output_66;
	::T_ROB_1:ABB_Library_Rob_1.PROFINET_Mapping_OUT.RTOOL_ROT_QUAT[2].OUTPUT[1] AT %QB."BASIC_V1_2".Module002_Output_67;
	::T_ROB_1:ABB_Library_Rob_1.PROFINET_Mapping_OUT.RTOOL_ROT_QUAT[2].OUTPUT[2] AT %QB."BASIC_V1_2".Module002_Output_68;
	::T_ROB_1:ABB_Library_Rob_1.PROFINET_Mapping_OUT.RTOOL_ROT_QUAT[2].OUTPUT[3] AT %QB."BASIC_V1_2".Module002_Output_69;
	::T_ROB_1:ABB_Library_Rob_1.PROFINET_Mapping_OUT.RTOOL_ROT_QUAT[3].OUTPUT[0] AT %QB."BASIC_V1_2".Module002_Output_70;
	::T_ROB_1:ABB_Library_Rob_1.PROFINET_Mapping_OUT.RTOOL_ROT_QUAT[3].OUTPUT[1] AT %QB."BASIC_V1_2".Module002_Output_71;
	::T_ROB_1:ABB_Library_Rob_1.PROFINET_Mapping_OUT.RTOOL_ROT_QUAT[3].OUTPUT[2] AT %QB."BASIC_V1_2".Module002_Output_72;
	::T_ROB_1:ABB_Library_Rob_1.PROFINET_Mapping_OUT.RTOOL_ROT_QUAT[3].OUTPUT[3] AT %QB."BASIC_V1_2".Module002_Output_73;
	::T_ROB_1:ABB_Library_Rob_1.PROFINET_Mapping_OUT.RTOOL_ROT_QUAT_SIGN.OUTPUT AT %QB."BASIC_V1_2".Module002_Output_74;
	::T_ROB_1:ABB_Library_Rob_1.PROFINET_Mapping_OUT.RTOOL_MASS.OUTPUT[0] AT %QB."BASIC_V1_2".Module002_Output_75;
	::T_ROB_1:ABB_Library_Rob_1.PROFINET_Mapping_OUT.RTOOL_MASS.OUTPUT[1] AT %QB."BASIC_V1_2".Module002_Output_76;
	::T_ROB_1:ABB_Library_Rob_1.PROFINET_Mapping_OUT.RTOOL_COG[0].OUTPUT[0] AT %QB."BASIC_V1_2".Module002_Output_77;
	::T_ROB_1:ABB_Library_Rob_1.PROFINET_Mapping_OUT.RTOOL_COG[0].OUTPUT[1] AT %QB."BASIC_V1_2".Module002_Output_78;
	::T_ROB_1:ABB_Library_Rob_1.PROFINET_Mapping_OUT.RTOOL_COG[0].OUTPUT[2] AT %QB."BASIC_V1_2".Module002_Output_79;
	::T_ROB_1:ABB_Library_Rob_1.PROFINET_Mapping_OUT.RTOOL_COG[0].OUTPUT[3] AT %QB."BASIC_V1_2".Module002_Output_80;
	::T_ROB_1:ABB_Library_Rob_1.PROFINET_Mapping_OUT.RTOOL_COG[1].OUTPUT[0] AT %QB."BASIC_V1_2".Module002_Output_81;
	::T_ROB_1:ABB_Library_Rob_1.PROFINET_Mapping_OUT.RTOOL_COG[1].OUTPUT[1] AT %QB."BASIC_V1_2".Module002_Output_82;
	::T_ROB_1:ABB_Library_Rob_1.PROFINET_Mapping_OUT.RTOOL_COG[1].OUTPUT[2] AT %QB."BASIC_V1_2".Module002_Output_83;
	::T_ROB_1:ABB_Library_Rob_1.PROFINET_Mapping_OUT.RTOOL_COG[1].OUTPUT[3] AT %QB."BASIC_V1_2".Module002_Output_84;
	::T_ROB_1:ABB_Library_Rob_1.PROFINET_Mapping_OUT.RTOOL_COG[2].OUTPUT[0] AT %QB."BASIC_V1_2".Module002_Output_85;
	::T_ROB_1:ABB_Library_Rob_1.PROFINET_Mapping_OUT.RTOOL_COG[2].OUTPUT[1] AT %QB."BASIC_V1_2".Module002_Output_86;
	::T_ROB_1:ABB_Library_Rob_1.PROFINET_Mapping_OUT.RTOOL_COG[2].OUTPUT[2] AT %QB."BASIC_V1_2".Module002_Output_87;
	::T_ROB_1:ABB_Library_Rob_1.PROFINET_Mapping_OUT.RTOOL_COG[2].OUTPUT[3] AT %QB."BASIC_V1_2".Module002_Output_88;
	::T_ROB_1:ABB_Library_Rob_1.PROFINET_Mapping_OUT.RTOOL_COG_SIGN.OUTPUT AT %QB."BASIC_V1_2".Module002_Output_89;
	::T_ROB_1:ABB_Library_Rob_1.PROFINET_Mapping_OUT.RTOOL_AOM_QUAT[0].OUTPUT[0] AT %QB."BASIC_V1_2".Module002_Output_90;
	::T_ROB_1:ABB_Library_Rob_1.PROFINET_Mapping_OUT.RTOOL_AOM_QUAT[0].OUTPUT[1] AT %QB."BASIC_V1_2".Module002_Output_91;
	::T_ROB_1:ABB_Library_Rob_1.PROFINET_Mapping_OUT.RTOOL_AOM_QUAT[0].OUTPUT[2] AT %QB."BASIC_V1_2".Module002_Output_92;
	::T_ROB_1:ABB_Library_Rob_1.PROFINET_Mapping_OUT.RTOOL_AOM_QUAT[0].OUTPUT[3] AT %QB."BASIC_V1_2".Module002_Output_93;
	::T_ROB_1:ABB_Library_Rob_1.PROFINET_Mapping_OUT.RTOOL_AOM_QUAT[1].OUTPUT[0] AT %QB."BASIC_V1_2".Module002_Output_94;
	::T_ROB_1:ABB_Library_Rob_1.PROFINET_Mapping_OUT.RTOOL_AOM_QUAT[1].OUTPUT[1] AT %QB."BASIC_V1_2".Module002_Output_95;
	::T_ROB_1:ABB_Library_Rob_1.PROFINET_Mapping_OUT.RTOOL_AOM_QUAT[1].OUTPUT[2] AT %QB."BASIC_V1_2".Module002_Output_96;
	::T_ROB_1:ABB_Library_Rob_1.PROFINET_Mapping_OUT.RTOOL_AOM_QUAT[1].OUTPUT[3] AT %QB."BASIC_V1_2".Module002_Output_97;
	::T_ROB_1:ABB_Library_Rob_1.PROFINET_Mapping_OUT.RTOOL_AOM_QUAT[2].OUTPUT[0] AT %QB."BASIC_V1_2".Module002_Output_98;
	::T_ROB_1:ABB_Library_Rob_1.PROFINET_Mapping_OUT.RTOOL_AOM_QUAT[2].OUTPUT[1] AT %QB."BASIC_V1_2".Module002_Output_99;
	::T_ROB_1:ABB_Library_Rob_1.PROFINET_Mapping_OUT.RTOOL_AOM_QUAT[2].OUTPUT[2] AT %QB."BASIC_V1_2".Module002_Output_100;
	::T_ROB_1:ABB_Library_Rob_1.PROFINET_Mapping_OUT.RTOOL_AOM_QUAT[2].OUTPUT[3] AT %QB."BASIC_V1_2".Module002_Output_101;
	::T_ROB_1:ABB_Library_Rob_1.PROFINET_Mapping_OUT.RTOOL_AOM_QUAT[3].OUTPUT[0] AT %QB."BASIC_V1_2".Module002_Output_102;
	::T_ROB_1:ABB_Library_Rob_1.PROFINET_Mapping_OUT.RTOOL_AOM_QUAT[3].OUTPUT[1] AT %QB."BASIC_V1_2".Module002_Output_103;
	::T_ROB_1:ABB_Library_Rob_1.PROFINET_Mapping_OUT.RTOOL_AOM_QUAT[3].OUTPUT[2] AT %QB."BASIC_V1_2".Module002_Output_104;
	::T_ROB_1:ABB_Library_Rob_1.PROFINET_Mapping_OUT.RTOOL_AOM_QUAT[3].OUTPUT[3] AT %QB."BASIC_V1_2".Module002_Output_105;
	::T_ROB_1:ABB_Library_Rob_1.PROFINET_Mapping_OUT.RTOOL_AOM_QUAT_SIGN.OUTPUT AT %QB."BASIC_V1_2".Module002_Output_106;
	::T_ROB_1:ABB_Library_Rob_1.PROFINET_Mapping_OUT.RTOOL_MOI[0].OUTPUT[0] AT %QB."BASIC_V1_2".Module002_Output_107;
	::T_ROB_1:ABB_Library_Rob_1.PROFINET_Mapping_OUT.RTOOL_MOI[0].OUTPUT[1] AT %QB."BASIC_V1_2".Module002_Output_108;
	::T_ROB_1:ABB_Library_Rob_1.PROFINET_Mapping_OUT.RTOOL_MOI[0].OUTPUT[2] AT %QB."BASIC_V1_2".Module002_Output_109;
	::T_ROB_1:ABB_Library_Rob_1.PROFINET_Mapping_OUT.RTOOL_MOI[0].OUTPUT[3] AT %QB."BASIC_V1_2".Module002_Output_110;
	::T_ROB_1:ABB_Library_Rob_1.PROFINET_Mapping_OUT.RTOOL_MOI[1].OUTPUT[0] AT %QB."BASIC_V1_2".Module002_Output_111;
	::T_ROB_1:ABB_Library_Rob_1.PROFINET_Mapping_OUT.RTOOL_MOI[1].OUTPUT[1] AT %QB."BASIC_V1_2".Module002_Output_112;
	::T_ROB_1:ABB_Library_Rob_1.PROFINET_Mapping_OUT.RTOOL_MOI[1].OUTPUT[2] AT %QB."BASIC_V1_2".Module002_Output_113;
	::T_ROB_1:ABB_Library_Rob_1.PROFINET_Mapping_OUT.RTOOL_MOI[1].OUTPUT[3] AT %QB."BASIC_V1_2".Module002_Output_114;
	::T_ROB_1:ABB_Library_Rob_1.PROFINET_Mapping_OUT.RTOOL_MOI[2].OUTPUT[0] AT %QB."BASIC_V1_2".Module002_Output_115;
	::T_ROB_1:ABB_Library_Rob_1.PROFINET_Mapping_OUT.RTOOL_MOI[2].OUTPUT[1] AT %QB."BASIC_V1_2".Module002_Output_116;
	::T_ROB_1:ABB_Library_Rob_1.PROFINET_Mapping_OUT.RTOOL_MOI[2].OUTPUT[2] AT %QB."BASIC_V1_2".Module002_Output_117;
	::T_ROB_1:ABB_Library_Rob_1.PROFINET_Mapping_OUT.RTOOL_MOI[2].OUTPUT[3] AT %QB."BASIC_V1_2".Module002_Output_118;
	::Global_T_ROB_2_PROFINET.Module_OK AT %IX."BASIC_V1_2a".ModuleOk;
	::T_ROB_2_L:ABB_Library_Rob_1.PROFINET_Mapping_IN.STATUS.INPUT AT %IB."BASIC_V1_2a".Module001_Input_0;
	::T_ROB_2_L:ABB_Library_Rob_1.PROFINET_Mapping_IN.SYSTEM.INPUT AT %IB."BASIC_V1_2a".Module001_Input_1;
	::T_ROB_2_L:ABB_Library_Rob_1.PROFINET_Mapping_IN.STATE_uID AT %IB."BASIC_V1_2a".Module001_Input_2;
	::T_ROB_2_L:ABB_Library_Rob_1.PROFINET_Mapping_IN.STATE_mID AT %IB."BASIC_V1_2a".Module001_Input_3;
	::T_ROB_2_L:ABB_Library_Rob_1.PROFINET_Mapping_IN.MOTION_TRAJECTORY_ID.INPUT[0] AT %IB."BASIC_V1_2a".Module001_Input_4;
	::T_ROB_2_L:ABB_Library_Rob_1.PROFINET_Mapping_IN.MOTION_TRAJECTORY_ID.INPUT[1] AT %IB."BASIC_V1_2a".Module001_Input_5;
	::T_ROB_2_L:ABB_Library_Rob_1.PROFINET_Mapping_IN.JOINT_POS[0].INPUT[0] AT %IB."BASIC_V1_2a".Module001_Input_6;
	::T_ROB_2_L:ABB_Library_Rob_1.PROFINET_Mapping_IN.JOINT_POS[0].INPUT[1] AT %IB."BASIC_V1_2a".Module001_Input_7;
	::T_ROB_2_L:ABB_Library_Rob_1.PROFINET_Mapping_IN.JOINT_POS[1].INPUT[0] AT %IB."BASIC_V1_2a".Module001_Input_8;
	::T_ROB_2_L:ABB_Library_Rob_1.PROFINET_Mapping_IN.JOINT_POS[1].INPUT[1] AT %IB."BASIC_V1_2a".Module001_Input_9;
	::T_ROB_2_L:ABB_Library_Rob_1.PROFINET_Mapping_IN.JOINT_POS[2].INPUT[0] AT %IB."BASIC_V1_2a".Module001_Input_10;
	::T_ROB_2_L:ABB_Library_Rob_1.PROFINET_Mapping_IN.JOINT_POS[2].INPUT[1] AT %IB."BASIC_V1_2a".Module001_Input_11;
	::T_ROB_2_L:ABB_Library_Rob_1.PROFINET_Mapping_IN.JOINT_POS[3].INPUT[0] AT %IB."BASIC_V1_2a".Module001_Input_12;
	::T_ROB_2_L:ABB_Library_Rob_1.PROFINET_Mapping_IN.JOINT_POS[3].INPUT[1] AT %IB."BASIC_V1_2a".Module001_Input_13;
	::T_ROB_2_L:ABB_Library_Rob_1.PROFINET_Mapping_IN.JOINT_POS[4].INPUT[0] AT %IB."BASIC_V1_2a".Module001_Input_14;
	::T_ROB_2_L:ABB_Library_Rob_1.PROFINET_Mapping_IN.JOINT_POS[4].INPUT[1] AT %IB."BASIC_V1_2a".Module001_Input_15;
	::T_ROB_2_L:ABB_Library_Rob_1.PROFINET_Mapping_IN.JOINT_POS[5].INPUT[0] AT %IB."BASIC_V1_2a".Module001_Input_16;
	::T_ROB_2_L:ABB_Library_Rob_1.PROFINET_Mapping_IN.JOINT_POS[5].INPUT[1] AT %IB."BASIC_V1_2a".Module001_Input_17;
	::T_ROB_2_L:ABB_Library_Rob_1.PROFINET_Mapping_IN.JOINT_POS[6].INPUT[0] AT %IB."BASIC_V1_2a".Module001_Input_18;
	::T_ROB_2_L:ABB_Library_Rob_1.PROFINET_Mapping_IN.JOINT_POS[6].INPUT[1] AT %IB."BASIC_V1_2a".Module001_Input_19;
	::T_ROB_2_L:ABB_Library_Rob_1.PROFINET_Mapping_IN.JOINT_POS_SIGN.INPUT AT %IB."BASIC_V1_2a".Module001_Input_20;
	::T_ROB_2_L:ABB_Library_Rob_1.PROFINET_Mapping_IN.TCP_POS[0].INPUT[0] AT %IB."BASIC_V1_2a".Module001_Input_21;
	::T_ROB_2_L:ABB_Library_Rob_1.PROFINET_Mapping_IN.TCP_POS[0].INPUT[1] AT %IB."BASIC_V1_2a".Module001_Input_22;
	::T_ROB_2_L:ABB_Library_Rob_1.PROFINET_Mapping_IN.TCP_POS[0].INPUT[2] AT %IB."BASIC_V1_2a".Module001_Input_23;
	::T_ROB_2_L:ABB_Library_Rob_1.PROFINET_Mapping_IN.TCP_POS[0].INPUT[3] AT %IB."BASIC_V1_2a".Module001_Input_24;
	::T_ROB_2_L:ABB_Library_Rob_1.PROFINET_Mapping_IN.TCP_POS[1].INPUT[0] AT %IB."BASIC_V1_2a".Module001_Input_25;
	::T_ROB_2_L:ABB_Library_Rob_1.PROFINET_Mapping_IN.TCP_POS[1].INPUT[1] AT %IB."BASIC_V1_2a".Module001_Input_26;
	::T_ROB_2_L:ABB_Library_Rob_1.PROFINET_Mapping_IN.TCP_POS[1].INPUT[2] AT %IB."BASIC_V1_2a".Module001_Input_27;
	::T_ROB_2_L:ABB_Library_Rob_1.PROFINET_Mapping_IN.TCP_POS[1].INPUT[3] AT %IB."BASIC_V1_2a".Module001_Input_28;
	::T_ROB_2_L:ABB_Library_Rob_1.PROFINET_Mapping_IN.TCP_POS[2].INPUT[0] AT %IB."BASIC_V1_2a".Module001_Input_29;
	::T_ROB_2_L:ABB_Library_Rob_1.PROFINET_Mapping_IN.TCP_POS[2].INPUT[1] AT %IB."BASIC_V1_2a".Module001_Input_30;
	::T_ROB_2_L:ABB_Library_Rob_1.PROFINET_Mapping_IN.TCP_POS[2].INPUT[2] AT %IB."BASIC_V1_2a".Module001_Input_31;
	::T_ROB_2_L:ABB_Library_Rob_1.PROFINET_Mapping_IN.TCP_POS[2].INPUT[3] AT %IB."BASIC_V1_2a".Module001_Input_32;
	::T_ROB_2_L:ABB_Library_Rob_1.PROFINET_Mapping_IN.TCP_ROT[0].INPUT[0] AT %IB."BASIC_V1_2a".Module001_Input_33;
	::T_ROB_2_L:ABB_Library_Rob_1.PROFINET_Mapping_IN.TCP_ROT[0].INPUT[1] AT %IB."BASIC_V1_2a".Module001_Input_34;
	::T_ROB_2_L:ABB_Library_Rob_1.PROFINET_Mapping_IN.TCP_ROT[1].INPUT[0] AT %IB."BASIC_V1_2a".Module001_Input_35;
	::T_ROB_2_L:ABB_Library_Rob_1.PROFINET_Mapping_IN.TCP_ROT[1].INPUT[1] AT %IB."BASIC_V1_2a".Module001_Input_36;
	::T_ROB_2_L:ABB_Library_Rob_1.PROFINET_Mapping_IN.TCP_ROT[2].INPUT[0] AT %IB."BASIC_V1_2a".Module001_Input_37;
	::T_ROB_2_L:ABB_Library_Rob_1.PROFINET_Mapping_IN.TCP_ROT[2].INPUT[1] AT %IB."BASIC_V1_2a".Module001_Input_38;
	::T_ROB_2_L:ABB_Library_Rob_1.PROFINET_Mapping_IN.TCP_EX_POS.INPUT[0] AT %IB."BASIC_V1_2a".Module001_Input_39;
	::T_ROB_2_L:ABB_Library_Rob_1.PROFINET_Mapping_IN.TCP_EX_POS.INPUT[1] AT %IB."BASIC_V1_2a".Module001_Input_40;
	::T_ROB_2_L:ABB_Library_Rob_1.PROFINET_Mapping_IN.TCP_SIGN.INPUT AT %IB."BASIC_V1_2a".Module001_Input_41;
	::T_ROB_2_L:ABB_Library_Rob_1.PROFINET_Mapping_IN.TCP_CFG[0] AT %IB."BASIC_V1_2a".Module001_Input_42;
	::T_ROB_2_L:ABB_Library_Rob_1.PROFINET_Mapping_IN.TCP_CFG[1] AT %IB."BASIC_V1_2a".Module001_Input_43;
	::T_ROB_2_L:ABB_Library_Rob_1.PROFINET_Mapping_IN.TCP_CFG[2] AT %IB."BASIC_V1_2a".Module001_Input_44;
	::T_ROB_2_L:ABB_Library_Rob_1.PROFINET_Mapping_IN.TCP_CFG[3] AT %IB."BASIC_V1_2a".Module001_Input_45;
	::T_ROB_2_L:ABB_Library_Rob_1.PROFINET_Mapping_IN.TCP_CFG_SIGN.INPUT AT %IB."BASIC_V1_2a".Module001_Input_46;
	::T_ROB_2_L:ABB_Library_Rob_1.PROFINET_Mapping_OUT.STATUS.OUTPUT AT %QB."BASIC_V1_2a".Module002_Output_0;
	::T_ROB_2_L:ABB_Library_Rob_1.PROFINET_Mapping_OUT.SYSTEM.OUTPUT AT %QB."BASIC_V1_2a".Module002_Output_1;
	::T_ROB_2_L:ABB_Library_Rob_1.PROFINET_Mapping_OUT.COMMAND.OUTPUT AT %QB."BASIC_V1_2a".Module002_Output_2;
	::T_ROB_2_L:ABB_Library_Rob_1.PROFINET_Mapping_OUT.COMMAND_mID AT %QB."BASIC_V1_2a".Module002_Output_3;
	::T_ROB_2_L:ABB_Library_Rob_1.PROFINET_Mapping_OUT.COMMAND_uID AT %QB."BASIC_V1_2a".Module002_Output_4;
	::T_ROB_2_L:ABB_Library_Rob_1.PROFINET_Mapping_OUT.TRAJECTORY_SIZE.OUTPUT[0] AT %QB."BASIC_V1_2a".Module002_Output_5;
	::T_ROB_2_L:ABB_Library_Rob_1.PROFINET_Mapping_OUT.TRAJECTORY_SIZE.OUTPUT[1] AT %QB."BASIC_V1_2a".Module002_Output_6;
	::T_ROB_2_L:ABB_Library_Rob_1.PROFINET_Mapping_OUT.SPEED AT %QB."BASIC_V1_2a".Module002_Output_7;
	::T_ROB_2_L:ABB_Library_Rob_1.PROFINET_Mapping_OUT.ZONE AT %QB."BASIC_V1_2a".Module002_Output_8;
	::T_ROB_2_L:ABB_Library_Rob_1.PROFINET_Mapping_OUT.JOINT_POS[0].OUTPUT[0] AT %QB."BASIC_V1_2a".Module002_Output_9;
	::T_ROB_2_L:ABB_Library_Rob_1.PROFINET_Mapping_OUT.JOINT_POS[0].OUTPUT[1] AT %QB."BASIC_V1_2a".Module002_Output_10;
	::T_ROB_2_L:ABB_Library_Rob_1.PROFINET_Mapping_OUT.JOINT_POS[1].OUTPUT[0] AT %QB."BASIC_V1_2a".Module002_Output_11;
	::T_ROB_2_L:ABB_Library_Rob_1.PROFINET_Mapping_OUT.JOINT_POS[1].OUTPUT[1] AT %QB."BASIC_V1_2a".Module002_Output_12;
	::T_ROB_2_L:ABB_Library_Rob_1.PROFINET_Mapping_OUT.JOINT_POS[2].OUTPUT[0] AT %QB."BASIC_V1_2a".Module002_Output_13;
	::T_ROB_2_L:ABB_Library_Rob_1.PROFINET_Mapping_OUT.JOINT_POS[2].OUTPUT[1] AT %QB."BASIC_V1_2a".Module002_Output_14;
	::T_ROB_2_L:ABB_Library_Rob_1.PROFINET_Mapping_OUT.JOINT_POS[3].OUTPUT[0] AT %QB."BASIC_V1_2a".Module002_Output_15;
	::T_ROB_2_L:ABB_Library_Rob_1.PROFINET_Mapping_OUT.JOINT_POS[3].OUTPUT[1] AT %QB."BASIC_V1_2a".Module002_Output_16;
	::T_ROB_2_L:ABB_Library_Rob_1.PROFINET_Mapping_OUT.JOINT_POS[4].OUTPUT[0] AT %QB."BASIC_V1_2a".Module002_Output_17;
	::T_ROB_2_L:ABB_Library_Rob_1.PROFINET_Mapping_OUT.JOINT_POS[4].OUTPUT[1] AT %QB."BASIC_V1_2a".Module002_Output_18;
	::T_ROB_2_L:ABB_Library_Rob_1.PROFINET_Mapping_OUT.JOINT_POS[5].OUTPUT[0] AT %QB."BASIC_V1_2a".Module002_Output_19;
	::T_ROB_2_L:ABB_Library_Rob_1.PROFINET_Mapping_OUT.JOINT_POS[5].OUTPUT[1] AT %QB."BASIC_V1_2a".Module002_Output_20;
	::T_ROB_2_L:ABB_Library_Rob_1.PROFINET_Mapping_OUT.JOINT_POS[6].OUTPUT[0] AT %QB."BASIC_V1_2a".Module002_Output_21;
	::T_ROB_2_L:ABB_Library_Rob_1.PROFINET_Mapping_OUT.JOINT_POS[6].OUTPUT[1] AT %QB."BASIC_V1_2a".Module002_Output_22;
	::T_ROB_2_L:ABB_Library_Rob_1.PROFINET_Mapping_OUT.JOINT_POS_SIGN.OUTPUT AT %QB."BASIC_V1_2a".Module002_Output_23;
	::T_ROB_2_L:ABB_Library_Rob_1.PROFINET_Mapping_OUT.TCP_POS[0].OUTPUT[0] AT %QB."BASIC_V1_2a".Module002_Output_24;
	::T_ROB_2_L:ABB_Library_Rob_1.PROFINET_Mapping_OUT.TCP_POS[0].OUTPUT[1] AT %QB."BASIC_V1_2a".Module002_Output_25;
	::T_ROB_2_L:ABB_Library_Rob_1.PROFINET_Mapping_OUT.TCP_POS[0].OUTPUT[2] AT %QB."BASIC_V1_2a".Module002_Output_26;
	::T_ROB_2_L:ABB_Library_Rob_1.PROFINET_Mapping_OUT.TCP_POS[0].OUTPUT[3] AT %QB."BASIC_V1_2a".Module002_Output_27;
	::T_ROB_2_L:ABB_Library_Rob_1.PROFINET_Mapping_OUT.TCP_POS[1].OUTPUT[0] AT %QB."BASIC_V1_2a".Module002_Output_28;
	::T_ROB_2_L:ABB_Library_Rob_1.PROFINET_Mapping_OUT.TCP_POS[1].OUTPUT[1] AT %QB."BASIC_V1_2a".Module002_Output_29;
	::T_ROB_2_L:ABB_Library_Rob_1.PROFINET_Mapping_OUT.TCP_POS[1].OUTPUT[2] AT %QB."BASIC_V1_2a".Module002_Output_30;
	::T_ROB_2_L:ABB_Library_Rob_1.PROFINET_Mapping_OUT.TCP_POS[1].OUTPUT[3] AT %QB."BASIC_V1_2a".Module002_Output_31;
	::T_ROB_2_L:ABB_Library_Rob_1.PROFINET_Mapping_OUT.TCP_POS[2].OUTPUT[0] AT %QB."BASIC_V1_2a".Module002_Output_32;
	::T_ROB_2_L:ABB_Library_Rob_1.PROFINET_Mapping_OUT.TCP_POS[2].OUTPUT[1] AT %QB."BASIC_V1_2a".Module002_Output_33;
	::T_ROB_2_L:ABB_Library_Rob_1.PROFINET_Mapping_OUT.TCP_POS[2].OUTPUT[2] AT %QB."BASIC_V1_2a".Module002_Output_34;
	::T_ROB_2_L:ABB_Library_Rob_1.PROFINET_Mapping_OUT.TCP_POS[2].OUTPUT[3] AT %QB."BASIC_V1_2a".Module002_Output_35;
	::T_ROB_2_L:ABB_Library_Rob_1.PROFINET_Mapping_OUT.TCP_ROT[0].OUTPUT[0] AT %QB."BASIC_V1_2a".Module002_Output_36;
	::T_ROB_2_L:ABB_Library_Rob_1.PROFINET_Mapping_OUT.TCP_ROT[0].OUTPUT[1] AT %QB."BASIC_V1_2a".Module002_Output_37;
	::T_ROB_2_L:ABB_Library_Rob_1.PROFINET_Mapping_OUT.TCP_ROT[1].OUTPUT[0] AT %QB."BASIC_V1_2a".Module002_Output_38;
	::T_ROB_2_L:ABB_Library_Rob_1.PROFINET_Mapping_OUT.TCP_ROT[1].OUTPUT[1] AT %QB."BASIC_V1_2a".Module002_Output_39;
	::T_ROB_2_L:ABB_Library_Rob_1.PROFINET_Mapping_OUT.TCP_ROT[2].OUTPUT[0] AT %QB."BASIC_V1_2a".Module002_Output_40;
	::T_ROB_2_L:ABB_Library_Rob_1.PROFINET_Mapping_OUT.TCP_ROT[2].OUTPUT[1] AT %QB."BASIC_V1_2a".Module002_Output_41;
	::T_ROB_2_L:ABB_Library_Rob_1.PROFINET_Mapping_OUT.TCP_EX_POS.OUTPUT[0] AT %QB."BASIC_V1_2a".Module002_Output_42;
	::T_ROB_2_L:ABB_Library_Rob_1.PROFINET_Mapping_OUT.TCP_EX_POS.OUTPUT[1] AT %QB."BASIC_V1_2a".Module002_Output_43;
	::T_ROB_2_L:ABB_Library_Rob_1.PROFINET_Mapping_OUT.TCP_SIGN.OUTPUT AT %QB."BASIC_V1_2a".Module002_Output_44;
	::T_ROB_2_L:ABB_Library_Rob_1.PROFINET_Mapping_OUT.TCP_CFG[0] AT %QB."BASIC_V1_2a".Module002_Output_45;
	::T_ROB_2_L:ABB_Library_Rob_1.PROFINET_Mapping_OUT.TCP_CFG[1] AT %QB."BASIC_V1_2a".Module002_Output_46;
	::T_ROB_2_L:ABB_Library_Rob_1.PROFINET_Mapping_OUT.TCP_CFG[2] AT %QB."BASIC_V1_2a".Module002_Output_47;
	::T_ROB_2_L:ABB_Library_Rob_1.PROFINET_Mapping_OUT.TCP_CFG[3] AT %QB."BASIC_V1_2a".Module002_Output_48;
	::T_ROB_2_L:ABB_Library_Rob_1.PROFINET_Mapping_OUT.TCP_CFG_SIGN.OUTPUT AT %QB."BASIC_V1_2a".Module002_Output_49;
	::T_ROB_2_L:ABB_Library_Rob_1.PROFINET_Mapping_OUT.RTOOL_RH.OUTPUT AT %QB."BASIC_V1_2a".Module002_Output_50;
	::T_ROB_2_L:ABB_Library_Rob_1.PROFINET_Mapping_OUT.RTOOL_POS[0].OUTPUT[0] AT %QB."BASIC_V1_2a".Module002_Output_51;
	::T_ROB_2_L:ABB_Library_Rob_1.PROFINET_Mapping_OUT.RTOOL_POS[0].OUTPUT[1] AT %QB."BASIC_V1_2a".Module002_Output_52;
	::T_ROB_2_L:ABB_Library_Rob_1.PROFINET_Mapping_OUT.RTOOL_POS[1].OUTPUT[0] AT %QB."BASIC_V1_2a".Module002_Output_53;
	::T_ROB_2_L:ABB_Library_Rob_1.PROFINET_Mapping_OUT.RTOOL_POS[1].OUTPUT[1] AT %QB."BASIC_V1_2a".Module002_Output_54;
	::T_ROB_2_L:ABB_Library_Rob_1.PROFINET_Mapping_OUT.RTOOL_POS[2].OUTPUT[0] AT %QB."BASIC_V1_2a".Module002_Output_55;
	::T_ROB_2_L:ABB_Library_Rob_1.PROFINET_Mapping_OUT.RTOOL_POS[2].OUTPUT[1] AT %QB."BASIC_V1_2a".Module002_Output_56;
	::T_ROB_2_L:ABB_Library_Rob_1.PROFINET_Mapping_OUT.RTOOL_POS_SIGN.OUTPUT AT %QB."BASIC_V1_2a".Module002_Output_57;
	::T_ROB_2_L:ABB_Library_Rob_1.PROFINET_Mapping_OUT.RTOOL_ROT_QUAT[0].OUTPUT[0] AT %QB."BASIC_V1_2a".Module002_Output_58;
	::T_ROB_2_L:ABB_Library_Rob_1.PROFINET_Mapping_OUT.RTOOL_ROT_QUAT[0].OUTPUT[1] AT %QB."BASIC_V1_2a".Module002_Output_59;
	::T_ROB_2_L:ABB_Library_Rob_1.PROFINET_Mapping_OUT.RTOOL_ROT_QUAT[0].OUTPUT[2] AT %QB."BASIC_V1_2a".Module002_Output_60;
	::T_ROB_2_L:ABB_Library_Rob_1.PROFINET_Mapping_OUT.RTOOL_ROT_QUAT[0].OUTPUT[3] AT %QB."BASIC_V1_2a".Module002_Output_61;
	::T_ROB_2_L:ABB_Library_Rob_1.PROFINET_Mapping_OUT.RTOOL_ROT_QUAT[1].OUTPUT[0] AT %QB."BASIC_V1_2a".Module002_Output_62;
	::T_ROB_2_L:ABB_Library_Rob_1.PROFINET_Mapping_OUT.RTOOL_ROT_QUAT[1].OUTPUT[1] AT %QB."BASIC_V1_2a".Module002_Output_63;
	::T_ROB_2_L:ABB_Library_Rob_1.PROFINET_Mapping_OUT.RTOOL_ROT_QUAT[1].OUTPUT[2] AT %QB."BASIC_V1_2a".Module002_Output_64;
	::T_ROB_2_L:ABB_Library_Rob_1.PROFINET_Mapping_OUT.RTOOL_ROT_QUAT[1].OUTPUT[3] AT %QB."BASIC_V1_2a".Module002_Output_65;
	::T_ROB_2_L:ABB_Library_Rob_1.PROFINET_Mapping_OUT.RTOOL_ROT_QUAT[2].OUTPUT[0] AT %QB."BASIC_V1_2a".Module002_Output_66;
	::T_ROB_2_L:ABB_Library_Rob_1.PROFINET_Mapping_OUT.RTOOL_ROT_QUAT[2].OUTPUT[1] AT %QB."BASIC_V1_2a".Module002_Output_67;
	::T_ROB_2_L:ABB_Library_Rob_1.PROFINET_Mapping_OUT.RTOOL_ROT_QUAT[2].OUTPUT[2] AT %QB."BASIC_V1_2a".Module002_Output_68;
	::T_ROB_2_L:ABB_Library_Rob_1.PROFINET_Mapping_OUT.RTOOL_ROT_QUAT[2].OUTPUT[3] AT %QB."BASIC_V1_2a".Module002_Output_69;
	::T_ROB_2_L:ABB_Library_Rob_1.PROFINET_Mapping_OUT.RTOOL_ROT_QUAT[3].OUTPUT[0] AT %QB."BASIC_V1_2a".Module002_Output_70;
	::T_ROB_2_L:ABB_Library_Rob_1.PROFINET_Mapping_OUT.RTOOL_ROT_QUAT[3].OUTPUT[1] AT %QB."BASIC_V1_2a".Module002_Output_71;
	::T_ROB_2_L:ABB_Library_Rob_1.PROFINET_Mapping_OUT.RTOOL_ROT_QUAT[3].OUTPUT[2] AT %QB."BASIC_V1_2a".Module002_Output_72;
	::T_ROB_2_L:ABB_Library_Rob_1.PROFINET_Mapping_OUT.RTOOL_ROT_QUAT[3].OUTPUT[3] AT %QB."BASIC_V1_2a".Module002_Output_73;
	::T_ROB_2_L:ABB_Library_Rob_1.PROFINET_Mapping_OUT.RTOOL_ROT_QUAT_SIGN.OUTPUT AT %QB."BASIC_V1_2a".Module002_Output_74;
	::T_ROB_2_L:ABB_Library_Rob_1.PROFINET_Mapping_OUT.RTOOL_MASS.OUTPUT[0] AT %QB."BASIC_V1_2a".Module002_Output_75;
	::T_ROB_2_L:ABB_Library_Rob_1.PROFINET_Mapping_OUT.RTOOL_MASS.OUTPUT[1] AT %QB."BASIC_V1_2a".Module002_Output_76;
	::T_ROB_2_L:ABB_Library_Rob_1.PROFINET_Mapping_OUT.RTOOL_COG[0].OUTPUT[0] AT %QB."BASIC_V1_2a".Module002_Output_77;
	::T_ROB_2_L:ABB_Library_Rob_1.PROFINET_Mapping_OUT.RTOOL_COG[0].OUTPUT[1] AT %QB."BASIC_V1_2a".Module002_Output_78;
	::T_ROB_2_L:ABB_Library_Rob_1.PROFINET_Mapping_OUT.RTOOL_COG[0].OUTPUT[2] AT %QB."BASIC_V1_2a".Module002_Output_79;
	::T_ROB_2_L:ABB_Library_Rob_1.PROFINET_Mapping_OUT.RTOOL_COG[0].OUTPUT[3] AT %QB."BASIC_V1_2a".Module002_Output_80;
	::T_ROB_2_L:ABB_Library_Rob_1.PROFINET_Mapping_OUT.RTOOL_COG[1].OUTPUT[0] AT %QB."BASIC_V1_2a".Module002_Output_81;
	::T_ROB_2_L:ABB_Library_Rob_1.PROFINET_Mapping_OUT.RTOOL_COG[1].OUTPUT[1] AT %QB."BASIC_V1_2a".Module002_Output_82;
	::T_ROB_2_L:ABB_Library_Rob_1.PROFINET_Mapping_OUT.RTOOL_COG[1].OUTPUT[2] AT %QB."BASIC_V1_2a".Module002_Output_83;
	::T_ROB_2_L:ABB_Library_Rob_1.PROFINET_Mapping_OUT.RTOOL_COG[1].OUTPUT[3] AT %QB."BASIC_V1_2a".Module002_Output_84;
	::T_ROB_2_L:ABB_Library_Rob_1.PROFINET_Mapping_OUT.RTOOL_COG[2].OUTPUT[0] AT %QB."BASIC_V1_2a".Module002_Output_85;
	::T_ROB_2_L:ABB_Library_Rob_1.PROFINET_Mapping_OUT.RTOOL_COG[2].OUTPUT[1] AT %QB."BASIC_V1_2a".Module002_Output_86;
	::T_ROB_2_L:ABB_Library_Rob_1.PROFINET_Mapping_OUT.RTOOL_COG[2].OUTPUT[2] AT %QB."BASIC_V1_2a".Module002_Output_87;
	::T_ROB_2_L:ABB_Library_Rob_1.PROFINET_Mapping_OUT.RTOOL_COG[2].OUTPUT[3] AT %QB."BASIC_V1_2a".Module002_Output_88;
	::T_ROB_2_L:ABB_Library_Rob_1.PROFINET_Mapping_OUT.RTOOL_COG_SIGN.OUTPUT AT %QB."BASIC_V1_2a".Module002_Output_89;
	::T_ROB_2_L:ABB_Library_Rob_1.PROFINET_Mapping_OUT.RTOOL_AOM_QUAT[0].OUTPUT[0] AT %QB."BASIC_V1_2a".Module002_Output_90;
	::T_ROB_2_L:ABB_Library_Rob_1.PROFINET_Mapping_OUT.RTOOL_AOM_QUAT[0].OUTPUT[1] AT %QB."BASIC_V1_2a".Module002_Output_91;
	::T_ROB_2_L:ABB_Library_Rob_1.PROFINET_Mapping_OUT.RTOOL_AOM_QUAT[0].OUTPUT[2] AT %QB."BASIC_V1_2a".Module002_Output_92;
	::T_ROB_2_L:ABB_Library_Rob_1.PROFINET_Mapping_OUT.RTOOL_AOM_QUAT[0].OUTPUT[3] AT %QB."BASIC_V1_2a".Module002_Output_93;
	::T_ROB_2_L:ABB_Library_Rob_1.PROFINET_Mapping_OUT.RTOOL_AOM_QUAT[1].OUTPUT[0] AT %QB."BASIC_V1_2a".Module002_Output_94;
	::T_ROB_2_L:ABB_Library_Rob_1.PROFINET_Mapping_OUT.RTOOL_AOM_QUAT[1].OUTPUT[1] AT %QB."BASIC_V1_2a".Module002_Output_95;
	::T_ROB_2_L:ABB_Library_Rob_1.PROFINET_Mapping_OUT.RTOOL_AOM_QUAT[1].OUTPUT[2] AT %QB."BASIC_V1_2a".Module002_Output_96;
	::T_ROB_2_L:ABB_Library_Rob_1.PROFINET_Mapping_OUT.RTOOL_AOM_QUAT[1].OUTPUT[3] AT %QB."BASIC_V1_2a".Module002_Output_97;
	::T_ROB_2_L:ABB_Library_Rob_1.PROFINET_Mapping_OUT.RTOOL_AOM_QUAT[2].OUTPUT[0] AT %QB."BASIC_V1_2a".Module002_Output_98;
	::T_ROB_2_L:ABB_Library_Rob_1.PROFINET_Mapping_OUT.RTOOL_AOM_QUAT[2].OUTPUT[1] AT %QB."BASIC_V1_2a".Module002_Output_99;
	::T_ROB_2_L:ABB_Library_Rob_1.PROFINET_Mapping_OUT.RTOOL_AOM_QUAT[2].OUTPUT[2] AT %QB."BASIC_V1_2a".Module002_Output_100;
	::T_ROB_2_L:ABB_Library_Rob_1.PROFINET_Mapping_OUT.RTOOL_AOM_QUAT[2].OUTPUT[3] AT %QB."BASIC_V1_2a".Module002_Output_101;
	::T_ROB_2_L:ABB_Library_Rob_1.PROFINET_Mapping_OUT.RTOOL_AOM_QUAT[3].OUTPUT[0] AT %QB."BASIC_V1_2a".Module002_Output_102;
	::T_ROB_2_L:ABB_Library_Rob_1.PROFINET_Mapping_OUT.RTOOL_AOM_QUAT[3].OUTPUT[1] AT %QB."BASIC_V1_2a".Module002_Output_103;
	::T_ROB_2_L:ABB_Library_Rob_1.PROFINET_Mapping_OUT.RTOOL_AOM_QUAT[3].OUTPUT[2] AT %QB."BASIC_V1_2a".Module002_Output_104;
	::T_ROB_2_L:ABB_Library_Rob_1.PROFINET_Mapping_OUT.RTOOL_AOM_QUAT[3].OUTPUT[3] AT %QB."BASIC_V1_2a".Module002_Output_105;
	::T_ROB_2_L:ABB_Library_Rob_1.PROFINET_Mapping_OUT.RTOOL_AOM_QUAT_SIGN.OUTPUT AT %QB."BASIC_V1_2a".Module002_Output_106;
	::T_ROB_2_L:ABB_Library_Rob_1.PROFINET_Mapping_OUT.RTOOL_MOI[0].OUTPUT[0] AT %QB."BASIC_V1_2a".Module002_Output_107;
	::T_ROB_2_L:ABB_Library_Rob_1.PROFINET_Mapping_OUT.RTOOL_MOI[0].OUTPUT[1] AT %QB."BASIC_V1_2a".Module002_Output_108;
	::T_ROB_2_L:ABB_Library_Rob_1.PROFINET_Mapping_OUT.RTOOL_MOI[0].OUTPUT[2] AT %QB."BASIC_V1_2a".Module002_Output_109;
	::T_ROB_2_L:ABB_Library_Rob_1.PROFINET_Mapping_OUT.RTOOL_MOI[0].OUTPUT[3] AT %QB."BASIC_V1_2a".Module002_Output_110;
	::T_ROB_2_L:ABB_Library_Rob_1.PROFINET_Mapping_OUT.RTOOL_MOI[1].OUTPUT[0] AT %QB."BASIC_V1_2a".Module002_Output_111;
	::T_ROB_2_L:ABB_Library_Rob_1.PROFINET_Mapping_OUT.RTOOL_MOI[1].OUTPUT[1] AT %QB."BASIC_V1_2a".Module002_Output_112;
	::T_ROB_2_L:ABB_Library_Rob_1.PROFINET_Mapping_OUT.RTOOL_MOI[1].OUTPUT[2] AT %QB."BASIC_V1_2a".Module002_Output_113;
	::T_ROB_2_L:ABB_Library_Rob_1.PROFINET_Mapping_OUT.RTOOL_MOI[1].OUTPUT[3] AT %QB."BASIC_V1_2a".Module002_Output_114;
	::T_ROB_2_L:ABB_Library_Rob_1.PROFINET_Mapping_OUT.RTOOL_MOI[2].OUTPUT[0] AT %QB."BASIC_V1_2a".Module002_Output_115;
	::T_ROB_2_L:ABB_Library_Rob_1.PROFINET_Mapping_OUT.RTOOL_MOI[2].OUTPUT[1] AT %QB."BASIC_V1_2a".Module002_Output_116;
	::T_ROB_2_L:ABB_Library_Rob_1.PROFINET_Mapping_OUT.RTOOL_MOI[2].OUTPUT[2] AT %QB."BASIC_V1_2a".Module002_Output_117;
	::T_ROB_2_L:ABB_Library_Rob_1.PROFINET_Mapping_OUT.RTOOL_MOI[2].OUTPUT[3] AT %QB."BASIC_V1_2a".Module002_Output_118;
	::T_ROB_2_R:ABB_Library_Rob_1.PROFINET_Mapping_IN.STATUS.INPUT AT %IB."BASIC_V1_2a".Module001_Input_128;
	::T_ROB_2_R:ABB_Library_Rob_1.PROFINET_Mapping_IN.SYSTEM.INPUT AT %IB."BASIC_V1_2a".Module001_Input_129;
	::T_ROB_2_R:ABB_Library_Rob_1.PROFINET_Mapping_IN.STATE_uID AT %IB."BASIC_V1_2a".Module001_Input_130;
	::T_ROB_2_R:ABB_Library_Rob_1.PROFINET_Mapping_IN.STATE_mID AT %IB."BASIC_V1_2a".Module001_Input_131;
	::T_ROB_2_R:ABB_Library_Rob_1.PROFINET_Mapping_IN.MOTION_TRAJECTORY_ID.INPUT[0] AT %IB."BASIC_V1_2a".Module001_Input_132;
	::T_ROB_2_R:ABB_Library_Rob_1.PROFINET_Mapping_IN.MOTION_TRAJECTORY_ID.INPUT[1] AT %IB."BASIC_V1_2a".Module001_Input_133;
	::T_ROB_2_R:ABB_Library_Rob_1.PROFINET_Mapping_IN.JOINT_POS[0].INPUT[0] AT %IB."BASIC_V1_2a".Module001_Input_134;
	::T_ROB_2_R:ABB_Library_Rob_1.PROFINET_Mapping_IN.JOINT_POS[0].INPUT[1] AT %IB."BASIC_V1_2a".Module001_Input_135;
	::T_ROB_2_R:ABB_Library_Rob_1.PROFINET_Mapping_IN.JOINT_POS[1].INPUT[0] AT %IB."BASIC_V1_2a".Module001_Input_136;
	::T_ROB_2_R:ABB_Library_Rob_1.PROFINET_Mapping_IN.JOINT_POS[1].INPUT[1] AT %IB."BASIC_V1_2a".Module001_Input_137;
	::T_ROB_2_R:ABB_Library_Rob_1.PROFINET_Mapping_IN.JOINT_POS[2].INPUT[0] AT %IB."BASIC_V1_2a".Module001_Input_138;
	::T_ROB_2_R:ABB_Library_Rob_1.PROFINET_Mapping_IN.JOINT_POS[2].INPUT[1] AT %IB."BASIC_V1_2a".Module001_Input_139;
	::T_ROB_2_R:ABB_Library_Rob_1.PROFINET_Mapping_IN.JOINT_POS[3].INPUT[0] AT %IB."BASIC_V1_2a".Module001_Input_140;
	::T_ROB_2_R:ABB_Library_Rob_1.PROFINET_Mapping_IN.JOINT_POS[3].INPUT[1] AT %IB."BASIC_V1_2a".Module001_Input_141;
	::T_ROB_2_R:ABB_Library_Rob_1.PROFINET_Mapping_IN.JOINT_POS[4].INPUT[0] AT %IB."BASIC_V1_2a".Module001_Input_142;
	::T_ROB_2_R:ABB_Library_Rob_1.PROFINET_Mapping_IN.JOINT_POS[4].INPUT[1] AT %IB."BASIC_V1_2a".Module001_Input_143;
	::T_ROB_2_R:ABB_Library_Rob_1.PROFINET_Mapping_IN.JOINT_POS[5].INPUT[0] AT %IB."BASIC_V1_2a".Module001_Input_144;
	::T_ROB_2_R:ABB_Library_Rob_1.PROFINET_Mapping_IN.JOINT_POS[5].INPUT[1] AT %IB."BASIC_V1_2a".Module001_Input_145;
	::T_ROB_2_R:ABB_Library_Rob_1.PROFINET_Mapping_IN.JOINT_POS[6].INPUT[0] AT %IB."BASIC_V1_2a".Module001_Input_146;
	::T_ROB_2_R:ABB_Library_Rob_1.PROFINET_Mapping_IN.JOINT_POS[6].INPUT[1] AT %IB."BASIC_V1_2a".Module001_Input_147;
	::T_ROB_2_R:ABB_Library_Rob_1.PROFINET_Mapping_IN.JOINT_POS_SIGN.INPUT AT %IB."BASIC_V1_2a".Module001_Input_148;
	::T_ROB_2_R:ABB_Library_Rob_1.PROFINET_Mapping_IN.TCP_POS[0].INPUT[0] AT %IB."BASIC_V1_2a".Module001_Input_149;
	::T_ROB_2_R:ABB_Library_Rob_1.PROFINET_Mapping_IN.TCP_POS[0].INPUT[1] AT %IB."BASIC_V1_2a".Module001_Input_150;
	::T_ROB_2_R:ABB_Library_Rob_1.PROFINET_Mapping_IN.TCP_POS[0].INPUT[2] AT %IB."BASIC_V1_2a".Module001_Input_151;
	::T_ROB_2_R:ABB_Library_Rob_1.PROFINET_Mapping_IN.TCP_POS[0].INPUT[3] AT %IB."BASIC_V1_2a".Module001_Input_152;
	::T_ROB_2_R:ABB_Library_Rob_1.PROFINET_Mapping_IN.TCP_POS[1].INPUT[0] AT %IB."BASIC_V1_2a".Module001_Input_153;
	::T_ROB_2_R:ABB_Library_Rob_1.PROFINET_Mapping_IN.TCP_POS[1].INPUT[1] AT %IB."BASIC_V1_2a".Module001_Input_154;
	::T_ROB_2_R:ABB_Library_Rob_1.PROFINET_Mapping_IN.TCP_POS[1].INPUT[2] AT %IB."BASIC_V1_2a".Module001_Input_155;
	::T_ROB_2_R:ABB_Library_Rob_1.PROFINET_Mapping_IN.TCP_POS[1].INPUT[3] AT %IB."BASIC_V1_2a".Module001_Input_156;
	::T_ROB_2_R:ABB_Library_Rob_1.PROFINET_Mapping_IN.TCP_POS[2].INPUT[0] AT %IB."BASIC_V1_2a".Module001_Input_157;
	::T_ROB_2_R:ABB_Library_Rob_1.PROFINET_Mapping_IN.TCP_POS[2].INPUT[1] AT %IB."BASIC_V1_2a".Module001_Input_158;
	::T_ROB_2_R:ABB_Library_Rob_1.PROFINET_Mapping_IN.TCP_POS[2].INPUT[2] AT %IB."BASIC_V1_2a".Module001_Input_159;
	::T_ROB_2_R:ABB_Library_Rob_1.PROFINET_Mapping_IN.TCP_POS[2].INPUT[3] AT %IB."BASIC_V1_2a".Module001_Input_160;
	::T_ROB_2_R:ABB_Library_Rob_1.PROFINET_Mapping_IN.TCP_ROT[0].INPUT[0] AT %IB."BASIC_V1_2a".Module001_Input_161;
	::T_ROB_2_R:ABB_Library_Rob_1.PROFINET_Mapping_IN.TCP_ROT[0].INPUT[1] AT %IB."BASIC_V1_2a".Module001_Input_162;
	::T_ROB_2_R:ABB_Library_Rob_1.PROFINET_Mapping_IN.TCP_ROT[1].INPUT[0] AT %IB."BASIC_V1_2a".Module001_Input_163;
	::T_ROB_2_R:ABB_Library_Rob_1.PROFINET_Mapping_IN.TCP_ROT[1].INPUT[1] AT %IB."BASIC_V1_2a".Module001_Input_164;
	::T_ROB_2_R:ABB_Library_Rob_1.PROFINET_Mapping_IN.TCP_ROT[2].INPUT[0] AT %IB."BASIC_V1_2a".Module001_Input_165;
	::T_ROB_2_R:ABB_Library_Rob_1.PROFINET_Mapping_IN.TCP_ROT[2].INPUT[1] AT %IB."BASIC_V1_2a".Module001_Input_166;
	::T_ROB_2_R:ABB_Library_Rob_1.PROFINET_Mapping_IN.TCP_EX_POS.INPUT[0] AT %IB."BASIC_V1_2a".Module001_Input_167;
	::T_ROB_2_R:ABB_Library_Rob_1.PROFINET_Mapping_IN.TCP_EX_POS.INPUT[1] AT %IB."BASIC_V1_2a".Module001_Input_168;
	::T_ROB_2_R:ABB_Library_Rob_1.PROFINET_Mapping_IN.TCP_SIGN.INPUT AT %IB."BASIC_V1_2a".Module001_Input_169;
	::T_ROB_2_R:ABB_Library_Rob_1.PROFINET_Mapping_IN.TCP_CFG[0] AT %IB."BASIC_V1_2a".Module001_Input_170;
	::T_ROB_2_R:ABB_Library_Rob_1.PROFINET_Mapping_IN.TCP_CFG[1] AT %IB."BASIC_V1_2a".Module001_Input_171;
	::T_ROB_2_R:ABB_Library_Rob_1.PROFINET_Mapping_IN.TCP_CFG[2] AT %IB."BASIC_V1_2a".Module001_Input_172;
	::T_ROB_2_R:ABB_Library_Rob_1.PROFINET_Mapping_IN.TCP_CFG[3] AT %IB."BASIC_V1_2a".Module001_Input_173;
	::T_ROB_2_R:ABB_Library_Rob_1.PROFINET_Mapping_IN.TCP_CFG_SIGN.INPUT AT %IB."BASIC_V1_2a".Module001_Input_174;
	::T_ROB_2_R:ABB_Library_Rob_1.PROFINET_Mapping_OUT.STATUS.OUTPUT AT %QB."BASIC_V1_2a".Module002_Output_128;
	::T_ROB_2_R:ABB_Library_Rob_1.PROFINET_Mapping_OUT.SYSTEM.OUTPUT AT %QB."BASIC_V1_2a".Module002_Output_129;
	::T_ROB_2_R:ABB_Library_Rob_1.PROFINET_Mapping_OUT.COMMAND.OUTPUT AT %QB."BASIC_V1_2a".Module002_Output_130;
	::T_ROB_2_R:ABB_Library_Rob_1.PROFINET_Mapping_OUT.COMMAND_mID AT %QB."BASIC_V1_2a".Module002_Output_131;
	::T_ROB_2_R:ABB_Library_Rob_1.PROFINET_Mapping_OUT.COMMAND_uID AT %QB."BASIC_V1_2a".Module002_Output_132;
	::T_ROB_2_R:ABB_Library_Rob_1.PROFINET_Mapping_OUT.TRAJECTORY_SIZE.OUTPUT[0] AT %QB."BASIC_V1_2a".Module002_Output_133;
	::T_ROB_2_R:ABB_Library_Rob_1.PROFINET_Mapping_OUT.TRAJECTORY_SIZE.OUTPUT[1] AT %QB."BASIC_V1_2a".Module002_Output_134;
	::T_ROB_2_R:ABB_Library_Rob_1.PROFINET_Mapping_OUT.SPEED AT %QB."BASIC_V1_2a".Module002_Output_135;
	::T_ROB_2_R:ABB_Library_Rob_1.PROFINET_Mapping_OUT.ZONE AT %QB."BASIC_V1_2a".Module002_Output_136;
	::T_ROB_2_R:ABB_Library_Rob_1.PROFINET_Mapping_OUT.JOINT_POS[0].OUTPUT[0] AT %QB."BASIC_V1_2a".Module002_Output_137;
	::T_ROB_2_R:ABB_Library_Rob_1.PROFINET_Mapping_OUT.JOINT_POS[0].OUTPUT[1] AT %QB."BASIC_V1_2a".Module002_Output_138;
	::T_ROB_2_R:ABB_Library_Rob_1.PROFINET_Mapping_OUT.JOINT_POS[1].OUTPUT[0] AT %QB."BASIC_V1_2a".Module002_Output_139;
	::T_ROB_2_R:ABB_Library_Rob_1.PROFINET_Mapping_OUT.JOINT_POS[1].OUTPUT[1] AT %QB."BASIC_V1_2a".Module002_Output_140;
	::T_ROB_2_R:ABB_Library_Rob_1.PROFINET_Mapping_OUT.JOINT_POS[2].OUTPUT[0] AT %QB."BASIC_V1_2a".Module002_Output_141;
	::T_ROB_2_R:ABB_Library_Rob_1.PROFINET_Mapping_OUT.JOINT_POS[2].OUTPUT[1] AT %QB."BASIC_V1_2a".Module002_Output_142;
	::T_ROB_2_R:ABB_Library_Rob_1.PROFINET_Mapping_OUT.JOINT_POS[3].OUTPUT[0] AT %QB."BASIC_V1_2a".Module002_Output_143;
	::T_ROB_2_R:ABB_Library_Rob_1.PROFINET_Mapping_OUT.JOINT_POS[3].OUTPUT[1] AT %QB."BASIC_V1_2a".Module002_Output_144;
	::T_ROB_2_R:ABB_Library_Rob_1.PROFINET_Mapping_OUT.JOINT_POS[4].OUTPUT[0] AT %QB."BASIC_V1_2a".Module002_Output_145;
	::T_ROB_2_R:ABB_Library_Rob_1.PROFINET_Mapping_OUT.JOINT_POS[4].OUTPUT[1] AT %QB."BASIC_V1_2a".Module002_Output_146;
	::T_ROB_2_R:ABB_Library_Rob_1.PROFINET_Mapping_OUT.JOINT_POS[5].OUTPUT[0] AT %QB."BASIC_V1_2a".Module002_Output_147;
	::T_ROB_2_R:ABB_Library_Rob_1.PROFINET_Mapping_OUT.JOINT_POS[5].OUTPUT[1] AT %QB."BASIC_V1_2a".Module002_Output_148;
	::T_ROB_2_R:ABB_Library_Rob_1.PROFINET_Mapping_OUT.JOINT_POS[6].OUTPUT[0] AT %QB."BASIC_V1_2a".Module002_Output_149;
	::T_ROB_2_R:ABB_Library_Rob_1.PROFINET_Mapping_OUT.JOINT_POS[6].OUTPUT[1] AT %QB."BASIC_V1_2a".Module002_Output_150;
	::T_ROB_2_R:ABB_Library_Rob_1.PROFINET_Mapping_OUT.JOINT_POS_SIGN.OUTPUT AT %QB."BASIC_V1_2a".Module002_Output_151;
	::T_ROB_2_R:ABB_Library_Rob_1.PROFINET_Mapping_OUT.TCP_POS[0].OUTPUT[0] AT %QB."BASIC_V1_2a".Module002_Output_152;
	::T_ROB_2_R:ABB_Library_Rob_1.PROFINET_Mapping_OUT.TCP_POS[0].OUTPUT[1] AT %QB."BASIC_V1_2a".Module002_Output_153;
	::T_ROB_2_R:ABB_Library_Rob_1.PROFINET_Mapping_OUT.TCP_POS[0].OUTPUT[2] AT %QB."BASIC_V1_2a".Module002_Output_154;
	::T_ROB_2_R:ABB_Library_Rob_1.PROFINET_Mapping_OUT.TCP_POS[0].OUTPUT[3] AT %QB."BASIC_V1_2a".Module002_Output_155;
	::T_ROB_2_R:ABB_Library_Rob_1.PROFINET_Mapping_OUT.TCP_POS[1].OUTPUT[0] AT %QB."BASIC_V1_2a".Module002_Output_156;
	::T_ROB_2_R:ABB_Library_Rob_1.PROFINET_Mapping_OUT.TCP_POS[1].OUTPUT[1] AT %QB."BASIC_V1_2a".Module002_Output_157;
	::T_ROB_2_R:ABB_Library_Rob_1.PROFINET_Mapping_OUT.TCP_POS[1].OUTPUT[2] AT %QB."BASIC_V1_2a".Module002_Output_158;
	::T_ROB_2_R:ABB_Library_Rob_1.PROFINET_Mapping_OUT.TCP_POS[1].OUTPUT[3] AT %QB."BASIC_V1_2a".Module002_Output_159;
	::T_ROB_2_R:ABB_Library_Rob_1.PROFINET_Mapping_OUT.TCP_POS[2].OUTPUT[0] AT %QB."BASIC_V1_2a".Module002_Output_160;
	::T_ROB_2_R:ABB_Library_Rob_1.PROFINET_Mapping_OUT.TCP_POS[2].OUTPUT[1] AT %QB."BASIC_V1_2a".Module002_Output_161;
	::T_ROB_2_R:ABB_Library_Rob_1.PROFINET_Mapping_OUT.TCP_POS[2].OUTPUT[2] AT %QB."BASIC_V1_2a".Module002_Output_162;
	::T_ROB_2_R:ABB_Library_Rob_1.PROFINET_Mapping_OUT.TCP_POS[2].OUTPUT[3] AT %QB."BASIC_V1_2a".Module002_Output_163;
	::T_ROB_2_R:ABB_Library_Rob_1.PROFINET_Mapping_OUT.TCP_ROT[0].OUTPUT[0] AT %QB."BASIC_V1_2a".Module002_Output_164;
	::T_ROB_2_R:ABB_Library_Rob_1.PROFINET_Mapping_OUT.TCP_ROT[0].OUTPUT[1] AT %QB."BASIC_V1_2a".Module002_Output_165;
	::T_ROB_2_R:ABB_Library_Rob_1.PROFINET_Mapping_OUT.TCP_ROT[1].OUTPUT[0] AT %QB."BASIC_V1_2a".Module002_Output_166;
	::T_ROB_2_R:ABB_Library_Rob_1.PROFINET_Mapping_OUT.TCP_ROT[1].OUTPUT[1] AT %QB."BASIC_V1_2a".Module002_Output_167;
	::T_ROB_2_R:ABB_Library_Rob_1.PROFINET_Mapping_OUT.TCP_ROT[2].OUTPUT[0] AT %QB."BASIC_V1_2a".Module002_Output_168;
	::T_ROB_2_R:ABB_Library_Rob_1.PROFINET_Mapping_OUT.TCP_ROT[2].OUTPUT[1] AT %QB."BASIC_V1_2a".Module002_Output_169;
	::T_ROB_2_R:ABB_Library_Rob_1.PROFINET_Mapping_OUT.TCP_EX_POS.OUTPUT[0] AT %QB."BASIC_V1_2a".Module002_Output_170;
	::T_ROB_2_R:ABB_Library_Rob_1.PROFINET_Mapping_OUT.TCP_EX_POS.OUTPUT[1] AT %QB."BASIC_V1_2a".Module002_Output_171;
	::T_ROB_2_R:ABB_Library_Rob_1.PROFINET_Mapping_OUT.TCP_SIGN.OUTPUT AT %QB."BASIC_V1_2a".Module002_Output_172;
	::T_ROB_2_R:ABB_Library_Rob_1.PROFINET_Mapping_OUT.TCP_CFG[0] AT %QB."BASIC_V1_2a".Module002_Output_173;
	::T_ROB_2_R:ABB_Library_Rob_1.PROFINET_Mapping_OUT.TCP_CFG[1] AT %QB."BASIC_V1_2a".Module002_Output_174;
	::T_ROB_2_R:ABB_Library_Rob_1.PROFINET_Mapping_OUT.TCP_CFG[2] AT %QB."BASIC_V1_2a".Module002_Output_175;
	::T_ROB_2_R:ABB_Library_Rob_1.PROFINET_Mapping_OUT.TCP_CFG[3] AT %QB."BASIC_V1_2a".Module002_Output_176;
	::T_ROB_2_R:ABB_Library_Rob_1.PROFINET_Mapping_OUT.TCP_CFG_SIGN.OUTPUT AT %QB."BASIC_V1_2a".Module002_Output_177;
	::T_ROB_2_R:ABB_Library_Rob_1.PROFINET_Mapping_OUT.RTOOL_RH.OUTPUT AT %QB."BASIC_V1_2a".Module002_Output_178;
	::T_ROB_2_R:ABB_Library_Rob_1.PROFINET_Mapping_OUT.RTOOL_POS[0].OUTPUT[0] AT %QB."BASIC_V1_2a".Module002_Output_179;
	::T_ROB_2_R:ABB_Library_Rob_1.PROFINET_Mapping_OUT.RTOOL_POS[0].OUTPUT[1] AT %QB."BASIC_V1_2a".Module002_Output_180;
	::T_ROB_2_R:ABB_Library_Rob_1.PROFINET_Mapping_OUT.RTOOL_POS[1].OUTPUT[0] AT %QB."BASIC_V1_2a".Module002_Output_181;
	::T_ROB_2_R:ABB_Library_Rob_1.PROFINET_Mapping_OUT.RTOOL_POS[1].OUTPUT[1] AT %QB."BASIC_V1_2a".Module002_Output_182;
	::T_ROB_2_R:ABB_Library_Rob_1.PROFINET_Mapping_OUT.RTOOL_POS[2].OUTPUT[0] AT %QB."BASIC_V1_2a".Module002_Output_183;
	::T_ROB_2_R:ABB_Library_Rob_1.PROFINET_Mapping_OUT.RTOOL_POS[2].OUTPUT[1] AT %QB."BASIC_V1_2a".Module002_Output_184;
	::T_ROB_2_R:ABB_Library_Rob_1.PROFINET_Mapping_OUT.RTOOL_POS_SIGN.OUTPUT AT %QB."BASIC_V1_2a".Module002_Output_185;
	::T_ROB_2_R:ABB_Library_Rob_1.PROFINET_Mapping_OUT.RTOOL_ROT_QUAT[0].OUTPUT[0] AT %QB."BASIC_V1_2a".Module002_Output_186;
	::T_ROB_2_R:ABB_Library_Rob_1.PROFINET_Mapping_OUT.RTOOL_ROT_QUAT[0].OUTPUT[1] AT %QB."BASIC_V1_2a".Module002_Output_187;
	::T_ROB_2_R:ABB_Library_Rob_1.PROFINET_Mapping_OUT.RTOOL_ROT_QUAT[0].OUTPUT[2] AT %QB."BASIC_V1_2a".Module002_Output_188;
	::T_ROB_2_R:ABB_Library_Rob_1.PROFINET_Mapping_OUT.RTOOL_ROT_QUAT[0].OUTPUT[3] AT %QB."BASIC_V1_2a".Module002_Output_189;
	::T_ROB_2_R:ABB_Library_Rob_1.PROFINET_Mapping_OUT.RTOOL_ROT_QUAT[1].OUTPUT[0] AT %QB."BASIC_V1_2a".Module002_Output_190;
	::T_ROB_2_R:ABB_Library_Rob_1.PROFINET_Mapping_OUT.RTOOL_ROT_QUAT[1].OUTPUT[1] AT %QB."BASIC_V1_2a".Module002_Output_191;
	::T_ROB_2_R:ABB_Library_Rob_1.PROFINET_Mapping_OUT.RTOOL_ROT_QUAT[1].OUTPUT[2] AT %QB."BASIC_V1_2a".Module002_Output_192;
	::T_ROB_2_R:ABB_Library_Rob_1.PROFINET_Mapping_OUT.RTOOL_ROT_QUAT[1].OUTPUT[3] AT %QB."BASIC_V1_2a".Module002_Output_193;
	::T_ROB_2_R:ABB_Library_Rob_1.PROFINET_Mapping_OUT.RTOOL_ROT_QUAT[2].OUTPUT[0] AT %QB."BASIC_V1_2a".Module002_Output_194;
	::T_ROB_2_R:ABB_Library_Rob_1.PROFINET_Mapping_OUT.RTOOL_ROT_QUAT[2].OUTPUT[1] AT %QB."BASIC_V1_2a".Module002_Output_195;
	::T_ROB_2_R:ABB_Library_Rob_1.PROFINET_Mapping_OUT.RTOOL_ROT_QUAT[2].OUTPUT[2] AT %QB."BASIC_V1_2a".Module002_Output_196;
	::T_ROB_2_R:ABB_Library_Rob_1.PROFINET_Mapping_OUT.RTOOL_ROT_QUAT[2].OUTPUT[3] AT %QB."BASIC_V1_2a".Module002_Output_197;
	::T_ROB_2_R:ABB_Library_Rob_1.PROFINET_Mapping_OUT.RTOOL_ROT_QUAT[3].OUTPUT[0] AT %QB."BASIC_V1_2a".Module002_Output_198;
	::T_ROB_2_R:ABB_Library_Rob_1.PROFINET_Mapping_OUT.RTOOL_ROT_QUAT[3].OUTPUT[1] AT %QB."BASIC_V1_2a".Module002_Output_199;
	::T_ROB_2_R:ABB_Library_Rob_1.PROFINET_Mapping_OUT.RTOOL_ROT_QUAT[3].OUTPUT[2] AT %QB."BASIC_V1_2a".Module002_Output_200;
	::T_ROB_2_R:ABB_Library_Rob_1.PROFINET_Mapping_OUT.RTOOL_ROT_QUAT[3].OUTPUT[3] AT %QB."BASIC_V1_2a".Module002_Output_201;
	::T_ROB_2_R:ABB_Library_Rob_1.PROFINET_Mapping_OUT.RTOOL_ROT_QUAT_SIGN.OUTPUT AT %QB."BASIC_V1_2a".Module002_Output_202;
	::T_ROB_2_R:ABB_Library_Rob_1.PROFINET_Mapping_OUT.RTOOL_MASS.OUTPUT[0] AT %QB."BASIC_V1_2a".Module002_Output_203;
	::T_ROB_2_R:ABB_Library_Rob_1.PROFINET_Mapping_OUT.RTOOL_MASS.OUTPUT[1] AT %QB."BASIC_V1_2a".Module002_Output_204;
	::T_ROB_2_R:ABB_Library_Rob_1.PROFINET_Mapping_OUT.RTOOL_COG[0].OUTPUT[0] AT %QB."BASIC_V1_2a".Module002_Output_205;
	::T_ROB_2_R:ABB_Library_Rob_1.PROFINET_Mapping_OUT.RTOOL_COG[0].OUTPUT[1] AT %QB."BASIC_V1_2a".Module002_Output_206;
	::T_ROB_2_R:ABB_Library_Rob_1.PROFINET_Mapping_OUT.RTOOL_COG[0].OUTPUT[2] AT %QB."BASIC_V1_2a".Module002_Output_207;
	::T_ROB_2_R:ABB_Library_Rob_1.PROFINET_Mapping_OUT.RTOOL_COG[0].OUTPUT[3] AT %QB."BASIC_V1_2a".Module002_Output_208;
	::T_ROB_2_R:ABB_Library_Rob_1.PROFINET_Mapping_OUT.RTOOL_COG[1].OUTPUT[0] AT %QB."BASIC_V1_2a".Module002_Output_209;
	::T_ROB_2_R:ABB_Library_Rob_1.PROFINET_Mapping_OUT.RTOOL_COG[1].OUTPUT[1] AT %QB."BASIC_V1_2a".Module002_Output_210;
	::T_ROB_2_R:ABB_Library_Rob_1.PROFINET_Mapping_OUT.RTOOL_COG[1].OUTPUT[2] AT %QB."BASIC_V1_2a".Module002_Output_211;
	::T_ROB_2_R:ABB_Library_Rob_1.PROFINET_Mapping_OUT.RTOOL_COG[1].OUTPUT[3] AT %QB."BASIC_V1_2a".Module002_Output_212;
	::T_ROB_2_R:ABB_Library_Rob_1.PROFINET_Mapping_OUT.RTOOL_COG[2].OUTPUT[0] AT %QB."BASIC_V1_2a".Module002_Output_213;
	::T_ROB_2_R:ABB_Library_Rob_1.PROFINET_Mapping_OUT.RTOOL_COG[2].OUTPUT[1] AT %QB."BASIC_V1_2a".Module002_Output_214;
	::T_ROB_2_R:ABB_Library_Rob_1.PROFINET_Mapping_OUT.RTOOL_COG[2].OUTPUT[2] AT %QB."BASIC_V1_2a".Module002_Output_215;
	::T_ROB_2_R:ABB_Library_Rob_1.PROFINET_Mapping_OUT.RTOOL_COG[2].OUTPUT[3] AT %QB."BASIC_V1_2a".Module002_Output_216;
	::T_ROB_2_R:ABB_Library_Rob_1.PROFINET_Mapping_OUT.RTOOL_COG_SIGN.OUTPUT AT %QB."BASIC_V1_2a".Module002_Output_217;
	::T_ROB_2_R:ABB_Library_Rob_1.PROFINET_Mapping_OUT.RTOOL_AOM_QUAT[0].OUTPUT[0] AT %QB."BASIC_V1_2a".Module002_Output_218;
	::T_ROB_2_R:ABB_Library_Rob_1.PROFINET_Mapping_OUT.RTOOL_AOM_QUAT[0].OUTPUT[1] AT %QB."BASIC_V1_2a".Module002_Output_219;
	::T_ROB_2_R:ABB_Library_Rob_1.PROFINET_Mapping_OUT.RTOOL_AOM_QUAT[0].OUTPUT[2] AT %QB."BASIC_V1_2a".Module002_Output_220;
	::T_ROB_2_R:ABB_Library_Rob_1.PROFINET_Mapping_OUT.RTOOL_AOM_QUAT[0].OUTPUT[3] AT %QB."BASIC_V1_2a".Module002_Output_221;
	::T_ROB_2_R:ABB_Library_Rob_1.PROFINET_Mapping_OUT.RTOOL_AOM_QUAT[1].OUTPUT[0] AT %QB."BASIC_V1_2a".Module002_Output_222;
	::T_ROB_2_R:ABB_Library_Rob_1.PROFINET_Mapping_OUT.RTOOL_AOM_QUAT[1].OUTPUT[1] AT %QB."BASIC_V1_2a".Module002_Output_223;
	::T_ROB_2_R:ABB_Library_Rob_1.PROFINET_Mapping_OUT.RTOOL_AOM_QUAT[1].OUTPUT[2] AT %QB."BASIC_V1_2a".Module002_Output_224;
	::T_ROB_2_R:ABB_Library_Rob_1.PROFINET_Mapping_OUT.RTOOL_AOM_QUAT[1].OUTPUT[3] AT %QB."BASIC_V1_2a".Module002_Output_225;
	::T_ROB_2_R:ABB_Library_Rob_1.PROFINET_Mapping_OUT.RTOOL_AOM_QUAT[2].OUTPUT[0] AT %QB."BASIC_V1_2a".Module002_Output_226;
	::T_ROB_2_R:ABB_Library_Rob_1.PROFINET_Mapping_OUT.RTOOL_AOM_QUAT[2].OUTPUT[1] AT %QB."BASIC_V1_2a".Module002_Output_227;
	::T_ROB_2_R:ABB_Library_Rob_1.PROFINET_Mapping_OUT.RTOOL_AOM_QUAT[2].OUTPUT[2] AT %QB."BASIC_V1_2a".Module002_Output_228;
	::T_ROB_2_R:ABB_Library_Rob_1.PROFINET_Mapping_OUT.RTOOL_AOM_QUAT[2].OUTPUT[3] AT %QB."BASIC_V1_2a".Module002_Output_229;
	::T_ROB_2_R:ABB_Library_Rob_1.PROFINET_Mapping_OUT.RTOOL_AOM_QUAT[3].OUTPUT[0] AT %QB."BASIC_V1_2a".Module002_Output_230;
	::T_ROB_2_R:ABB_Library_Rob_1.PROFINET_Mapping_OUT.RTOOL_AOM_QUAT[3].OUTPUT[1] AT %QB."BASIC_V1_2a".Module002_Output_231;
	::T_ROB_2_R:ABB_Library_Rob_1.PROFINET_Mapping_OUT.RTOOL_AOM_QUAT[3].OUTPUT[2] AT %QB."BASIC_V1_2a".Module002_Output_232;
	::T_ROB_2_R:ABB_Library_Rob_1.PROFINET_Mapping_OUT.RTOOL_AOM_QUAT[3].OUTPUT[3] AT %QB."BASIC_V1_2a".Module002_Output_233;
	::T_ROB_2_R:ABB_Library_Rob_1.PROFINET_Mapping_OUT.RTOOL_AOM_QUAT_SIGN.OUTPUT AT %QB."BASIC_V1_2a".Module002_Output_234;
	::T_ROB_2_R:ABB_Library_Rob_1.PROFINET_Mapping_OUT.RTOOL_MOI[0].OUTPUT[0] AT %QB."BASIC_V1_2a".Module002_Output_235;
	::T_ROB_2_R:ABB_Library_Rob_1.PROFINET_Mapping_OUT.RTOOL_MOI[0].OUTPUT[1] AT %QB."BASIC_V1_2a".Module002_Output_236;
	::T_ROB_2_R:ABB_Library_Rob_1.PROFINET_Mapping_OUT.RTOOL_MOI[0].OUTPUT[2] AT %QB."BASIC_V1_2a".Module002_Output_237;
	::T_ROB_2_R:ABB_Library_Rob_1.PROFINET_Mapping_OUT.RTOOL_MOI[0].OUTPUT[3] AT %QB."BASIC_V1_2a".Module002_Output_238;
	::T_ROB_2_R:ABB_Library_Rob_1.PROFINET_Mapping_OUT.RTOOL_MOI[1].OUTPUT[0] AT %QB."BASIC_V1_2a".Module002_Output_239;
	::T_ROB_2_R:ABB_Library_Rob_1.PROFINET_Mapping_OUT.RTOOL_MOI[1].OUTPUT[1] AT %QB."BASIC_V1_2a".Module002_Output_240;
	::T_ROB_2_R:ABB_Library_Rob_1.PROFINET_Mapping_OUT.RTOOL_MOI[1].OUTPUT[2] AT %QB."BASIC_V1_2a".Module002_Output_241;
	::T_ROB_2_R:ABB_Library_Rob_1.PROFINET_Mapping_OUT.RTOOL_MOI[1].OUTPUT[3] AT %QB."BASIC_V1_2a".Module002_Output_242;
	::T_ROB_2_R:ABB_Library_Rob_1.PROFINET_Mapping_OUT.RTOOL_MOI[2].OUTPUT[0] AT %QB."BASIC_V1_2a".Module002_Output_243;
	::T_ROB_2_R:ABB_Library_Rob_1.PROFINET_Mapping_OUT.RTOOL_MOI[2].OUTPUT[1] AT %QB."BASIC_V1_2a".Module002_Output_244;
	::T_ROB_2_R:ABB_Library_Rob_1.PROFINET_Mapping_OUT.RTOOL_MOI[2].OUTPUT[2] AT %QB."BASIC_V1_2a".Module002_Output_245;
	::T_ROB_2_R:ABB_Library_Rob_1.PROFINET_Mapping_OUT.RTOOL_MOI[2].OUTPUT[3] AT %QB."BASIC_V1_2a".Module002_Output_246;
END_VAR
```

- Safety project (password-protected, skipped)

### Cfg_mMot.axis - 5APC2100_BY48_000/mappMotion/Cfg_mMot.axis
```
Element gAxis_Mech_01 (Type=axis)
  BaseTypeIsReadOnly = 0
  BaseType = LinearBounded
    MeasurementUnit = 5066068
    MeasurementResolutionIsReadOnly = 0
    MeasurementResolution = 0.01
    CountDirectionIsReadOnly = 0
    CountDirection = Inverse
  MovementLimitsIsReadOnly = 0
  MovementLimits = Internal
    Position:
      LowerLimitMin = -1.79769313486231E308
      UpperLimitMax = 1.79769313486231E308
      LowerLimit = -4
      UpperLimit = 1402
    VelocityIsReadOnly = 0
    Velocity:
      VelocityMax = 3.4E38
      Velocity = 2000
    AccelerationIsReadOnly = 0
    Acceleration:
      AccelerationMax = 3.4E38
      Acceleration = 20000
    DecelerationIsReadOnly = 0
    Deceleration:
      DecelerationMax = 3.4E38
      Deceleration = 20000
  Alarms = None
Element gAxis_Mech_02 (Type=axis)
  BaseTypeIsReadOnly = 0
  BaseType = LinearBounded
    MeasurementUnit = 5066068
    MeasurementResolutionIsReadOnly = 0
    MeasurementResolution = 0.01
    CountDirectionIsReadOnly = 0
    CountDirection = Inverse
  MovementLimitsIsReadOnly = 0
  MovementLimits = Internal
    Position:
      LowerLimitMin = -1.79769313486231E308
      UpperLimitMax = 1.79769313486231E308
      LowerLimit = -4
      UpperLimit = 1402
    VelocityIsReadOnly = 0
    Velocity:
      VelocityMax = 3.4E38
      Velocity = 2000
    AccelerationIsReadOnly = 0
    Acceleration:
      AccelerationMax = 3.4E38
      Acceleration = 20000
    DecelerationIsReadOnly = 0
    Deceleration:
      DecelerationMax = 3.4E38
      Deceleration = 20000
  Alarms = None
Element gAxis_ROB_01 (Type=axis)
  BaseTypeIsReadOnly = 0
  BaseType = LinearBounded
    MeasurementUnit = 5066068
    MeasurementResolutionIsReadOnly = 0
    MeasurementResolution = 0.01
    CountDirectionIsReadOnly = 0
    CountDirection = Standard
  MovementLimitsIsReadOnly = 0
  MovementLimits = Internal
    Position:
      LowerLimitMin = -1.79769313486231E308
      UpperLimitMax = 1.79769313486231E308
      LowerLimit = -4
      UpperLimit = 802
    VelocityIsReadOnly = 0
    Velocity:
      VelocityMax = 3.4E38
      Velocity = 500
    AccelerationIsReadOnly = 0
    Acceleration:
      AccelerationMax = 3.4E38
      Acceleration = 5000
    DecelerationIsReadOnly = 0
    Deceleration:
      DecelerationMax = 3.4E38
      Deceleration = 5000
  Alarms = None
```

## Logical view

Binary libraries used (declarations not repeated): operator, runtime, astime, AsIecCon, AsZip, FileIO, AsSafety, standard, DataObj, AsXml, McBase 5.26.1, MpBase, MpAxis 5.26.1, McAcpPar 5.26.1, McAcpAx 5.26.1, McAxis 5.26.1, McAxGroup 5.26.1, CoTrace 5.24.1

### Global.typ - Global data types
```iecst
TYPE
	T_ROB_2_PROFINET_Str : 	STRUCT
		Module_OK : BOOL;
	END_STRUCT;
	VInRoS_Str : 	STRUCT
		Mech_Id_1 : Mechanism_Str;
		Mech_Id_2 : Mechanism_Str;
		Mech_Id_3 : Mechanism_Str;
		Rob_Id_1 : Robot_Str;
		Rob_Id_2_L : Robot_Str;
		Rob_Id_2_R : Robot_Str;
		EX_600 : EX_600_Str;
	END_STRUCT;
	Mechanism_Str : 	STRUCT
		Command : Mechanism_Command_Str;
		Info : Mechanism_Info_Str;
		Parameters : Mechanism_Parameters_Str;
		Position : LREAL;
	END_STRUCT;
	Mechanism_Command_Str : 	STRUCT
		Power : BOOL;
		Home : BOOL;
		Start : BOOL;
		Stop : BOOL;
		Reset_Error : BOOL;
		Reset_Safety : BOOL;
		Update : BOOL;
		Move : BOOL;
	END_STRUCT;
	Mechanism_Info_Str : 	STRUCT
		Active : BOOL;
		Power : BOOL;
		Home : BOOL;
		Safety : BOOL;
		Error : BOOL;
		In_Position : BOOL;
		Update_Done : BOOL;
		Move_Active : BOOL;
	END_STRUCT;
	Mechanism_Parameters_Str : 	STRUCT
		Position : LREAL;
		Velocity : REAL;
		Acc_Dec : REAL;
	END_STRUCT;
	EX_600_Str : 	STRUCT
		Slave : EX_600_Slave_Str;
	END_STRUCT;
	EX_600_Slave_Str : 	STRUCT
		Command : EX_600_Command_Str;
		Info : EX_600_Info_Str;
		Input : ARRAY[0..15]OF BOOL;
		Output : ARRAY[0..7]OF BOOL;
	END_STRUCT;
	EX_600_Command_Str : 	STRUCT
		Home : BOOL;
		Reset_Error : BOOL;
	END_STRUCT;
	EX_600_Info_Str : 	STRUCT
		Active : BOOL;
		Home : BOOL;
		Error : BOOL;
	END_STRUCT;
	Robot_Str : 	STRUCT
		Command : Robot_Command_Str;
		Info : Robot_Info_Str;
		Position : Robot_Position_Str;
	END_STRUCT;
	Robot_Command_Str : 	STRUCT
		Power : BOOL;
		Home : BOOL;
		Start : BOOL;
		Stop : BOOL;
		Reset_Error : BOOL;
		Reset_Safety : BOOL;
	END_STRUCT;
	Robot_Info_Str : 	STRUCT
		Active : BOOL;
		Power : BOOL;
		Home : BOOL;
		Safety : BOOL;
		Error : BOOL;
		In_Position : BOOL;
		Update_Done : BOOL;
		Move_Active : BOOL;
	END_STRUCT;
	Robot_Position_Str : 	STRUCT
		Q : ARRAY[0..6]OF REAL;
	END_STRUCT;
END_TYPE
```

### Global.var - Global variables
```iecst
VAR
	Global_VInRoS_Str : VInRoS_Str;
	RESET_SAFETY : BOOL;
	SAFETY_ACTIVE : BOOL;
	SAFETY_STATUS : BOOL;
	SIMULATION_ENABLE : BOOL := FALSE;
	ROB_1_Sim_PROFINET_Mapping_OUT : ARRAY[0..255] OF USINT;
	ROB_1_Sim_PROFINET_Mapping_IN : ARRAY[0..255] OF USINT;
	Global_T_ROB_2_PROFINET : T_ROB_2_PROFINET_Str;
END_VAR
```


### Program Logical/T_MECH_1 (ANSIC)

#### Main.h
```c
#include <bur/plctypes.h>

#ifdef _DEFAULT_INCLUDES
#include <AsDefault.h>
#endif

typedef enum Mechanism_State_ID_enum{
	MECH_STATE_ACTIVE,
	MECH_STATE_POWER,
	MECH_STATE_HOME,
	MECH_STATE_WAIT,
	MECH_STATE_UPD_PARAMETERS,
	MECH_STATE_MOTION_1,
	MECH_STATE_MOTION_2,
	MECH_STATE_HOME_UPD_PARAMETERS,
	MECH_STATE_HOME_MOTION_1,
	MECH_STATE_HOME_MOTION_2,
	MECH_STATE_STOP,
	MECH_STATE_SAFETY,
	MECH_STATE_ERROR
}Mechanism_State_ID_enum;
```

#### Main.c
```c
#include <bur/plctypes.h>

#ifdef _DEFAULT_INCLUDES
#include <AsDefault.h>
#endif

#include "Main.h"

_LOCAL struct MpAxisBasic MpAxisBasic_0;
_LOCAL struct MpAxisBasicParType AxisParameters;
_LOCAL enum Mechanism_State_ID_enum state_id;

void _INIT ProgramInit(void)
{
	memset(&Global_VInRoS_Str.Mech_Id_1, 0, sizeof(Global_VInRoS_Str.Mech_Id_1));

	AxisParameters.Homing.Mode = mcHOMING_ABSOLUTE;
	AxisParameters.Homing.Position = 1770365;

	MpAxisBasic_0.Enable     = 1;
	MpAxisBasic_0.MpLink     = &gAxis_Mech_01;
	MpAxisBasic_0.Parameters = &AxisParameters;

	Trajectory_Str.Targets.Position[0] = 100.0;
	Trajectory_Str.Targets.Position[1] = 1100.0;
	Trajectory_Str.Targets.Position[2] = 700.0;
	Trajectory_Str.Targets.Position[3] = 300.0;
	Trajectory_Str.Targets.Position[4] = 1200.0;

	Trajectory_Str.Targets.Velocity[0] = 500.0;
	Trajectory_Str.Targets.Velocity[1] = 1000.0;
	Trajectory_Str.Targets.Velocity[2] = 200.0;
	Trajectory_Str.Targets.Velocity[3] = 1500.0;
	Trajectory_Str.Targets.Velocity[4] = 400.0;

	Trajectory_Str.Length = 5;

	state_id = MECH_STATE_ACTIVE;
}

void _CYCLIC ProgramCyclic(void)
{
	switch(state_id){
		case MECH_STATE_ACTIVE:
			{
				if(Global_VInRoS_Str.Mech_Id_1.Info.Active == TRUE){
					state_id = MECH_STATE_POWER;
				}
			}
			break;

		case MECH_STATE_POWER:
			{
				if(Global_VInRoS_Str.Mech_Id_1.Info.Power == TRUE){
					state_id = MECH_STATE_HOME;
				}
			}
			break;

		case MECH_STATE_HOME:
			{
				if(Global_VInRoS_Str.Mech_Id_1.Info.Home == TRUE){
					MpAxisBasic_0.Home = FALSE;
					Global_VInRoS_Str.Mech_Id_1.Command.Home = FALSE;
					state_id = MECH_STATE_WAIT;
				}
			}
			break;

		case MECH_STATE_WAIT:
			{
				if(Global_VInRoS_Str.Mech_Id_1.Command.Home == TRUE){
					state_id = MECH_STATE_HOME_UPD_PARAMETERS;
				}

				if(Global_VInRoS_Str.Mech_Id_1.Command.Start == TRUE){
					Trajectory_Str.Iteration = 0;
					state_id = MECH_STATE_UPD_PARAMETERS;
				}
			}
			break;

		case MECH_STATE_UPD_PARAMETERS:
			{
				Global_VInRoS_Str.Mech_Id_1.Parameters.Position = Trajectory_Str.Targets.Position[Trajectory_Str.Iteration];
				Global_VInRoS_Str.Mech_Id_1.Parameters.Velocity = Trajectory_Str.Targets.Velocity[Trajectory_Str.Iteration];
				Global_VInRoS_Str.Mech_Id_1.Parameters.Acc_Dec  = Trajectory_Str.Targets.Velocity[Trajectory_Str.Iteration]*10;

				Global_VInRoS_Str.Mech_Id_1.Command.Update = TRUE;
				if(Global_VInRoS_Str.Mech_Id_1.Info.Update_Done == TRUE){
					state_id = MECH_STATE_MOTION_1;
				}
			}
			break;

		case MECH_STATE_MOTION_1:
			{
				Global_VInRoS_Str.Mech_Id_1.Command.Move = TRUE;
				if(Global_VInRoS_Str.Mech_Id_1.Info.Move_Active == TRUE){
					state_id = MECH_STATE_MOTION_2;
				}
			}
			break;

		case MECH_STATE_MOTION_2:
			{
				if(Global_VInRoS_Str.Mech_Id_1.Command.Stop == TRUE){
					state_id = MECH_STATE_STOP;
				}else{
					if(Global_VInRoS_Str.Mech_Id_1.Info.In_Position == TRUE){
						Global_VInRoS_Str.Mech_Id_1.Command.Move = 0;

						if(Trajectory_Str.Iteration == Trajectory_Str.Length - 1){
							state_id = MECH_STATE_WAIT;
						}else{
							Trajectory_Str.Iteration++;
							state_id = MECH_STATE_UPD_PARAMETERS;
						}
					}
				}
			}
			break;

		case MECH_STATE_HOME_UPD_PARAMETERS:
			{
				Global_VInRoS_Str.Mech_Id_1.Parameters.Position = 700.0;
				Global_VInRoS_Str.Mech_Id_1.Parameters.Velocity = 500.0;
				Global_VInRoS_Str.Mech_Id_1.Parameters.Acc_Dec  = 5000.0;

				Global_VInRoS_Str.Mech_Id_1.Command.Update = TRUE;
				if(Global_VInRoS_Str.Mech_Id_1.Info.Update_Done == TRUE){
					state_id = MECH_STATE_HOME_MOTION_1;
				}
			}
			break;

		case MECH_STATE_HOME_MOTION_1:
			{
				Global_VInRoS_Str.Mech_Id_1.Command.Move = TRUE;
				if(Global_VInRoS_Str.Mech_Id_1.Info.Move_Active == TRUE){
					state_id = MECH_STATE_HOME_MOTION_2;
				}
			}
			break;

		case MECH_STATE_HOME_MOTION_2:
			{
				if(Global_VInRoS_Str.Mech_Id_1.Info.In_Position == TRUE){
					Global_VInRoS_Str.Mech_Id_1.Command.Move = FALSE;
					Global_VInRoS_Str.Mech_Id_1.Command.Home = FALSE;
					state_id = MECH_STATE_WAIT;
				}
			}
			break;

		case MECH_STATE_STOP:
			{
				Global_VInRoS_Str.Mech_Id_1.Command.Stop  = FALSE;
				Global_VInRoS_Str.Mech_Id_1.Command.Start = FALSE;

				Global_VInRoS_Str.Mech_Id_1.Command.Move = FALSE;
				if(Global_VInRoS_Str.Mech_Id_1.Info.Move_Active == FALSE){
					state_id = MECH_STATE_WAIT;
				}
			}
			break;

		case MECH_STATE_SAFETY:
			{
			}
			break;

		case MECH_STATE_ERROR:
			{
				Global_VInRoS_Str.Mech_Id_1.Command.Home   = FALSE;
				Global_VInRoS_Str.Mech_Id_1.Command.Update = FALSE;
				Global_VInRoS_Str.Mech_Id_1.Command.Stop   = FALSE;
				Global_VInRoS_Str.Mech_Id_1.Command.Start  = FALSE;
				Global_VInRoS_Str.Mech_Id_1.Command.Move   = FALSE;

				if(Global_VInRoS_Str.Mech_Id_1.Info.Error == FALSE){
					state_id = MECH_STATE_WAIT;
				}
			}
			break;

	}

	AxisParameters.Position     = Global_VInRoS_Str.Mech_Id_1.Parameters.Position;
	AxisParameters.Velocity     = Global_VInRoS_Str.Mech_Id_1.Parameters.Velocity;
	AxisParameters.Acceleration = Global_VInRoS_Str.Mech_Id_1.Parameters.Acc_Dec;
	AxisParameters.Deceleration = Global_VInRoS_Str.Mech_Id_1.Parameters.Acc_Dec;

	MpAxisBasic_0.Power = Global_VInRoS_Str.Mech_Id_1.Command.Power;
	if(Global_VInRoS_Str.Mech_Id_1.Command.Home == TRUE && Global_VInRoS_Str.Mech_Id_1.Info.Home == FALSE){
		MpAxisBasic_0.Home = TRUE;
	}
	MpAxisBasic_0.ErrorReset = Global_VInRoS_Str.Mech_Id_1.Command.Reset_Error;
	MpAxisBasic_0.Update     = Global_VInRoS_Str.Mech_Id_1.Command.Update;
	MpAxisBasic_0.MoveAbsolute = Global_VInRoS_Str.Mech_Id_1.Command.Move;

	MpAxisBasic(&MpAxisBasic_0);

	Global_VInRoS_Str.Mech_Id_1.Info.Active = MpAxisBasic_0.Active;
	Global_VInRoS_Str.Mech_Id_1.Info.Power  = MpAxisBasic_0.PowerOn;
	Global_VInRoS_Str.Mech_Id_1.Info.Home   = MpAxisBasic_0.IsHomed;
	Global_VInRoS_Str.Mech_Id_1.Info.Error  = MpAxisBasic_0.Error;
	Global_VInRoS_Str.Mech_Id_1.Info.Update_Done = MpAxisBasic_0.UpdateDone;
	Global_VInRoS_Str.Mech_Id_1.Info.Move_Active = MpAxisBasic_0.MoveActive;
	if(MpAxisBasic_0.InPosition == TRUE && MpAxisBasic_0.MoveDone == TRUE){
		Global_VInRoS_Str.Mech_Id_1.Info.In_Position = TRUE;
	}else{
		Global_VInRoS_Str.Mech_Id_1.Info.In_Position = FALSE;
	}
	Global_VInRoS_Str.Mech_Id_1.Info.Safety = FALSE;

	Global_VInRoS_Str.Mech_Id_1.Position = MpAxisBasic_0.Position;

	if(Global_VInRoS_Str.Mech_Id_1.Info.Error == TRUE){
		state_id = MECH_STATE_ERROR;
	}
}
```

### Program Logical/T_MECH_2 (ANSIC)

#### Main.h
```c
#include <bur/plctypes.h>

#ifdef _DEFAULT_INCLUDES
#include <AsDefault.h>
#endif

typedef enum Mechanism_State_ID_enum{
	MECH_STATE_ACTIVE,
	MECH_STATE_POWER,
	MECH_STATE_HOME,
	MECH_STATE_WAIT,
	MECH_STATE_UPD_PARAMETERS,
	MECH_STATE_MOTION_1,
	MECH_STATE_MOTION_2,
	MECH_STATE_HOME_UPD_PARAMETERS,
	MECH_STATE_HOME_MOTION_1,
	MECH_STATE_HOME_MOTION_2,
	MECH_STATE_STOP,
	MECH_STATE_SAFETY,
	MECH_STATE_ERROR
}Mechanism_State_ID_enum;
```

#### Main.c
```c
#include <bur/plctypes.h>

#ifdef _DEFAULT_INCLUDES
#include <AsDefault.h>
#endif

#include "Main.h"

_LOCAL struct MpAxisBasic MpAxisBasic_0;
_LOCAL struct MpAxisBasicParType AxisParameters;
_LOCAL enum Mechanism_State_ID_enum state_id;

void _INIT ProgramInit(void)
{
	memset(&Global_VInRoS_Str.Mech_Id_2, 0, sizeof(Global_VInRoS_Str.Mech_Id_2));

	AxisParameters.Homing.Mode = mcHOMING_ABSOLUTE;
	AxisParameters.Homing.Position = 2219977;

	MpAxisBasic_0.Enable     = TRUE;
	MpAxisBasic_0.MpLink     = &gAxis_Mech_02;
	MpAxisBasic_0.Parameters = &AxisParameters;

	Trajectory_Str.Targets.Position[0] = 100.0;
	Trajectory_Str.Targets.Position[1] = 1100.0;
	Trajectory_Str.Targets.Position[2] = 700.0;
	Trajectory_Str.Targets.Position[3] = 200.0;
	Trajectory_Str.Targets.Position[4] = 1200.0;

	Trajectory_Str.Targets.Velocity[0] = 500.0;
	Trajectory_Str.Targets.Velocity[1] = 1000.0;
	Trajectory_Str.Targets.Velocity[2] = 200.0;
	Trajectory_Str.Targets.Velocity[3] = 500.0;
	Trajectory_Str.Targets.Velocity[4] = 400.0;

	Trajectory_Str.Length = 5;

	state_id = MECH_STATE_ACTIVE;
}

void _CYCLIC ProgramCyclic(void)
{
	if(SIMULATION_ENABLE == FALSE){
		switch(state_id){
			case MECH_STATE_ACTIVE:
				{
					if(Global_VInRoS_Str.Mech_Id_2.Info.Active == TRUE){
						state_id = MECH_STATE_POWER;
					}
				}
				break;

			case MECH_STATE_POWER:
				{
					if(Global_VInRoS_Str.Mech_Id_2.Info.Power == TRUE){
						state_id = MECH_STATE_HOME;
					}
				}
				break;

			case MECH_STATE_HOME:
				{
					if(Global_VInRoS_Str.Mech_Id_2.Info.Home == TRUE){
						MpAxisBasic_0.Home = FALSE;
						Global_VInRoS_Str.Mech_Id_2.Command.Home = FALSE;
						state_id = MECH_STATE_WAIT;
					}
				}
				break;

			case MECH_STATE_WAIT:
				{
					if(Global_VInRoS_Str.Mech_Id_2.Command.Home == TRUE){
						state_id = MECH_STATE_HOME_UPD_PARAMETERS;
					}

					if(Global_VInRoS_Str.Mech_Id_2.Command.Start == TRUE){
						Trajectory_Str.Iteration = FALSE;
						state_id = MECH_STATE_UPD_PARAMETERS;
					}
				}
				break;

			case MECH_STATE_UPD_PARAMETERS:
				{
					Global_VInRoS_Str.Mech_Id_2.Parameters.Position = Trajectory_Str.Targets.Position[Trajectory_Str.Iteration];
					Global_VInRoS_Str.Mech_Id_2.Parameters.Velocity = Trajectory_Str.Targets.Velocity[Trajectory_Str.Iteration];
					Global_VInRoS_Str.Mech_Id_2.Parameters.Acc_Dec  = Trajectory_Str.Targets.Velocity[Trajectory_Str.Iteration]*10;

					Global_VInRoS_Str.Mech_Id_2.Command.Update = TRUE;
					if(Global_VInRoS_Str.Mech_Id_2.Info.Update_Done == TRUE){
						state_id = MECH_STATE_MOTION_1;
					}
				}
				break;

			case MECH_STATE_MOTION_1:
				{
					Global_VInRoS_Str.Mech_Id_2.Command.Move = TRUE;
					if(Global_VInRoS_Str.Mech_Id_2.Info.Move_Active == TRUE){
						state_id = MECH_STATE_MOTION_2;
					}
				}
				break;

			case MECH_STATE_MOTION_2:
				{
					if(Global_VInRoS_Str.Mech_Id_2.Command.Stop == TRUE){
						state_id = MECH_STATE_STOP;
					}else{
						if(Global_VInRoS_Str.Mech_Id_2.Info.In_Position == TRUE){
							Global_VInRoS_Str.Mech_Id_2.Command.Move = FALSE;

							if(Trajectory_Str.Iteration == Trajectory_Str.Length - 1){
								state_id = MECH_STATE_WAIT;
							}else{
								Trajectory_Str.Iteration++;
								state_id = MECH_STATE_UPD_PARAMETERS;
							}
						}
					}
				}
				break;

			case MECH_STATE_HOME_UPD_PARAMETERS:
				{
					Global_VInRoS_Str.Mech_Id_2.Parameters.Position = 700.0;
					Global_VInRoS_Str.Mech_Id_2.Parameters.Velocity = 500.0;
					Global_VInRoS_Str.Mech_Id_2.Parameters.Acc_Dec  = 5000.0;

					Global_VInRoS_Str.Mech_Id_2.Command.Update = TRUE;
					if(Global_VInRoS_Str.Mech_Id_2.Info.Update_Done == TRUE){
						state_id = MECH_STATE_HOME_MOTION_1;
					}
				}
				break;

			case MECH_STATE_HOME_MOTION_1:
				{
					Global_VInRoS_Str.Mech_Id_2.Command.Move = TRUE;
					if(Global_VInRoS_Str.Mech_Id_2.Info.Move_Active == TRUE){
						state_id = MECH_STATE_HOME_MOTION_2;
					}
				}
				break;

			case MECH_STATE_HOME_MOTION_2:
				{
					if(Global_VInRoS_Str.Mech_Id_2.Info.In_Position == TRUE){
						Global_VInRoS_Str.Mech_Id_2.Command.Move = FALSE;
						Global_VInRoS_Str.Mech_Id_2.Command.Home = FALSE;
						state_id = MECH_STATE_WAIT;
					}
				}
				break;

			case MECH_STATE_STOP:
				{
					Global_VInRoS_Str.Mech_Id_2.Command.Stop  = FALSE;
					Global_VInRoS_Str.Mech_Id_2.Command.Start = FALSE;

					Global_VInRoS_Str.Mech_Id_2.Command.Move = FALSE;
					if(Global_VInRoS_Str.Mech_Id_2.Info.Move_Active == FALSE){
						state_id = MECH_STATE_WAIT;
					}
				}
				break;

			case MECH_STATE_SAFETY:
				{
				}
				break;

			case MECH_STATE_ERROR:
				{
					Global_VInRoS_Str.Mech_Id_2.Command.Home   = FALSE;
					Global_VInRoS_Str.Mech_Id_2.Command.Update = FALSE;
					Global_VInRoS_Str.Mech_Id_2.Command.Stop   = FALSE;
					Global_VInRoS_Str.Mech_Id_2.Command.Start  = FALSE;
					Global_VInRoS_Str.Mech_Id_2.Command.Move   = FALSE;

					Global_VInRoS_Str.Mech_Id_2.Command.Move = FALSE;
					if(Global_VInRoS_Str.Mech_Id_2.Info.Error == FALSE){
						state_id = MECH_STATE_WAIT;
					}
				}
				break;

		}

		AxisParameters.Position     = Global_VInRoS_Str.Mech_Id_2.Parameters.Position;
		AxisParameters.Velocity     = Global_VInRoS_Str.Mech_Id_2.Parameters.Velocity;
		AxisParameters.Acceleration = Global_VInRoS_Str.Mech_Id_2.Parameters.Acc_Dec;
		AxisParameters.Deceleration = Global_VInRoS_Str.Mech_Id_2.Parameters.Acc_Dec;

		MpAxisBasic_0.Power = Global_VInRoS_Str.Mech_Id_2.Command.Power;
		if(Global_VInRoS_Str.Mech_Id_2.Command.Home == TRUE && Global_VInRoS_Str.Mech_Id_2.Info.Home == FALSE){
			MpAxisBasic_0.Home = TRUE;
		}
		MpAxisBasic_0.ErrorReset = Global_VInRoS_Str.Mech_Id_2.Command.Reset_Error;
		MpAxisBasic_0.Update     = Global_VInRoS_Str.Mech_Id_2.Command.Update;
		MpAxisBasic_0.MoveAbsolute = Global_VInRoS_Str.Mech_Id_2.Command.Move;

		MpAxisBasic(&MpAxisBasic_0);

		Global_VInRoS_Str.Mech_Id_2.Info.Active = MpAxisBasic_0.Active;
		Global_VInRoS_Str.Mech_Id_2.Info.Power  = MpAxisBasic_0.PowerOn;
		Global_VInRoS_Str.Mech_Id_2.Info.Home   = MpAxisBasic_0.IsHomed;
		Global_VInRoS_Str.Mech_Id_2.Info.Error  = MpAxisBasic_0.Error;
		Global_VInRoS_Str.Mech_Id_2.Info.Update_Done = MpAxisBasic_0.UpdateDone;
		Global_VInRoS_Str.Mech_Id_2.Info.Move_Active = MpAxisBasic_0.MoveActive;
		if(MpAxisBasic_0.InPosition == TRUE && MpAxisBasic_0.MoveDone == TRUE){
			Global_VInRoS_Str.Mech_Id_2.Info.In_Position = TRUE;
		}else{
			Global_VInRoS_Str.Mech_Id_2.Info.In_Position = FALSE;
		}
		Global_VInRoS_Str.Mech_Id_2.Info.Safety = FALSE;

		Global_VInRoS_Str.Mech_Id_2.Position = MpAxisBasic_0.Position;

		if(Global_VInRoS_Str.Mech_Id_2.Info.Error == TRUE){
			state_id = MECH_STATE_ERROR;
		}
	}else{
		switch(state_id){
			case MECH_STATE_ACTIVE:
				{
					if(Global_VInRoS_Str.Mech_Id_2.Info.Active == TRUE){
						state_id = MECH_STATE_WAIT;
					}
				}
				break;

			case MECH_STATE_WAIT:
				{
					if(Global_VInRoS_Str.Mech_Id_2.Command.Home == TRUE && Global_VInRoS_Str.Mech_Id_2.Info.Move_Active == FALSE){
						state_id = MECH_STATE_HOME_MOTION_1;
					}

					if(Global_VInRoS_Str.Mech_Id_2.Command.Start == TRUE && Global_VInRoS_Str.Mech_Id_2.Info.Move_Active == FALSE){
						state_id = MECH_STATE_MOTION_1;
					}

					if(Global_VInRoS_Str.Mech_Id_2.Command.Stop == TRUE && Global_VInRoS_Str.Mech_Id_2.Info.Move_Active == TRUE){
						state_id = MECH_STATE_STOP;
					}

				}
				break;

			case MECH_STATE_MOTION_1:
				{
					if(Global_VInRoS_Str.Mech_Id_2.Info.Move_Active == TRUE){
						Global_VInRoS_Str.Mech_Id_2.Command.Start = FALSE;
						state_id = MECH_STATE_WAIT;
					}
				}
				break;

			case MECH_STATE_HOME_MOTION_1:
				{
					if(Global_VInRoS_Str.Mech_Id_2.Info.Move_Active == TRUE){
						Global_VInRoS_Str.Mech_Id_2.Command.Home = FALSE;
						state_id = MECH_STATE_WAIT;
					}
				}
				break;

			case MECH_STATE_STOP:
				{
					if(Global_VInRoS_Str.Mech_Id_2.Info.Move_Active == FALSE){
						Global_VInRoS_Str.Mech_Id_2.Command.Stop = FALSE;
						state_id = MECH_STATE_WAIT;
					}
				}
				break;
		}

		Global_VInRoS_Str.Mech_Id_2.Info.Power = TRUE;
		Global_VInRoS_Str.Mech_Id_2.Info.Home  = TRUE;
	}
}
```

### Program Logical/T_MECH_3 (ANSIC)
